// TwinCAT 3 PLC project SchrauberAblauf_SK
// ProgramVersion: 3.1.4024.0
// libraries:
//   Tc2_MC2, * (Beckhoff Automation GmbH)
//   Tc2_Standard, * (Beckhoff Automation GmbH)
//   Tc2_System, * (Beckhoff Automation GmbH)
//   Tc2_Utilities, * (Beckhoff Automation GmbH)
//   Tc3_Module, * (Beckhoff Automation GmbH)
//   UniLib Gruppe 11, * (Beckhoff Automation GmbH & Co. KG)
//   UniNc Gruppe 11, * (Beckhoff Automation GmbH & Co. KG)
//   VisuSymbols,3.5.10.0,System
// project tree:
//   DUTs/ ST_MeldServoSchrauber_1.TcDUT (not stored), ST_ParamSKSServoschrauber.TcDUT (not stored), ST_SKSSchrauberInOut_Vis.TcDUT
//   / GlobalTextList.TcGTLO, PlcTask.TcTTO (not stored), TL_AuswahlSchrauberAblauf.TcTLO, Visualisierungsmanager.TcVMO (not stored)
//   GVLs/ GlobalVar_InOut.TcGVL, GlobalVar_Constant.TcGVL, GlobalVar_NcAchsen.TcGVL, GVL_VISU_SCHRAUBER.TcGVL
//   POUs/10_Funktionen/Diverse/ FB_AchsStartAusf.TcPOU, FB_ErrorCnt.TcPOU (not stored), FB_LogFile_Schrauber.TcPOU, FB_Mittelwert.TcPOU (not stored), FB_OBJ_TimeStamp.TcPOU, FB_Zeitstempel.TcPOU, F_Inbetween.TcPOU (not stored), F_PosZustand.TcPOU
//   POUs/10_Funktionen/History/ FB_StepHistory.TcPOU (not stored)
//   POUs/10_Funktionen/SchraubBearb/Obj/ FB_Obj_Error_Schrauber.TcPOU (not stored), FB_Obj_IOSchlauch.TcPOU
//   POUs/ MAIN.TcPOU, prgMAIN.TcPOU, PRG_Schrauber.TcPOU
//   POUs/SchrauberAblauf/ FB_Schrauber_PnP.TcPOU, FB_Schrauber_PnP_Neu_1.TcPOU
//   POUs/Simulationsprogramm/ FB_Schrauber_Simulation.TcPOU, PRG_Schrauber_Test.TcPOU
//   VISUs/ Frame_Schlauch_Bedien.TcVIS, Frame_Schrauber.TcVIS, Frame_Schrauber_Bedien.TcVIS, Frame_Schrauber_Status.TcVIS, Schrauber_Aufruf.TcVIS

// ---- DUTs/ST_SKSSchrauberInOut_Vis.TcDUT
TYPE ST_SKSSchrauberInOut_Vis :
STRUCT
	I_bTaktFrg						: BOOL;
	I_bTaktStop						: BOOL;
	I_bAuto							: BOOL;
	I_bHand							: BOOL;
	I_bQuittFehler					: BOOL;

	I_bTaktStart					: BOOL;	(*Start Schienenschrauben*)

	I_bGrdstlgSchrEinh				: BOOL;
	I_bZustellZylAusgef				: BOOL;

	I_fSchraubTiefeAuswurf			: LREAL;

	I_fTiefentoleranzPositiv		: LREAL:=1;	(* Z.B. 3 bedeutet, dass von Solltiefe bis + 3mm wir im Ziel liegen *)
	I_fTiefentoleranzNegativ		: LREAL:=0.5;	(* Z.B. 3 bedeutet, dass von Solltiefe bis - 3mm wir im Ziel liegen *)
		
	I_bSchraubeNachschiessen		: BOOL;

	I_bFreigabeAuswerfen			: BOOL;
	
	I_bSchlauchBelegt				:BOOL;
	I_bSchrauberBelegt				:BOOL;
	I_bAuswurfStart					:BOOL;
	I_bVereinzelungStart			:BOOL;
	
	Q_bBusy							: BOOL;
	Q_bDone							: BOOL;
	Q_bError						: BOOL;
	
	Q_nErrorId						: INT;
	Q_bDrehmomentFehler				: BOOL;
	
	Q_bDrehmomentOk					:BOOL;
	
	Q_nActTorque					:LREAL; 	(* Drehmoment ausgabe Mittelwert *)
	Q_nActDepth						:LREAL; 	(* Tiefen ausgabe  *)
	Q_nActVelo						:LREAL;		
	Q_nActPos						:LREAL;
	
	Q_nLastTorque					:LREAL;
	Q_nLastDepth					:LREAL;
	
	Q_nStep							: INT;
	
	Q_strStep						: STRING;
	Q_sStatus						: STRING(255);	//Informationen zu dem aktuellen Ablaufschritt
	
END_STRUCT
END_TYPE

// ---- GVLs/GlobalVar_InOut.TcGVL
{attribute 'Tc2GvlVarNames'}
VAR_GLOBAL
	(* Inputs *)
	bGVLEndlageZyl_1_Eingef	AT %I*: BOOL;
	bGVLEndlageZyl_1_Ausgef	AT %I*: BOOL;
	
	bGVLEndlageZyl_2_Eingef	AT %I*: BOOL;
	bGVLEndlageZyl_2_Ausgef	AT %I*: BOOL;
	
	(* Outputs *)
	bGVLVentil_1_Ausfahr	AT %Q*: BOOL;
	bGVLVentil_1_Einfahr	AT %Q*: BOOL;
	
	bGVLVentil_2_Ausfahr	AT %Q*: BOOL;
	bGVLVentil_2_Einfahr	AT %Q*: BOOL;
	
END_VAR

// ---- GVLs/GlobalVar_Constant.TcGVL
{attribute 'Tc2GvlVarNames'}
VAR_GLOBAL CONSTANT
	cGrundPos								:INT :=1;
	cBearbPos								:INT :=3;
	
	cAxis1261_Schrauber1					:INT := 1;
	cEnc03_Schrauber1						:INT := 2;
	
END_VAR

// ---- GVLs/GlobalVar_NcAchsen.TcGVL
{attribute 'Tc2GvlVarNames'}
VAR_GLOBAL
	
	arrAxis									: ARRAY[1..2] OF AXIS_REF;
	arrNcAchsen								: ARRAY[1..2] OF  TC3_UniLib.ST_NcAchsen;		(* Achtung 1 = Achse / 2= Encoder für Tiefenmessung *)
	arrStartAusf							: ARRAY[1..2] OF FB_AchsStartAusf;
	arrAnstgSchrauberAchse					: ARRAY[1..2] OF FB_AchsKontrlAnstg;
	
	arrBetrartAutomAktiv					:ARRAY[1..2] OF BOOL;
	arrAntrGruppeFrg						:ARRAY[1..2] OF BOOL;
	stParamSKSServoschrauber				:ST_ParamSKSServoschrauber;
	
	objSchlauch								: FB_Obj_IOSchlauch;
	stAchsMeldung							: ST_MeldServoSchrauber_1;					
	bTakt2Langsam							:BOOL;
	
	
	
END_VAR

// ---- GVLs/GVL_VISU_SCHRAUBER.TcGVL
{attribute 'Tc2GvlVarNames'}
VAR_GLOBAL
	stSKSSchrauberInOut_Vis_Schr_1		:ST_SKSSchrauberInOut_Vis;
END_VAR

// ---- POUs/10_Funktionen/Diverse/FB_AchsStartAusf.TcPOU
FUNCTION_BLOCK FB_AchsStartAusf
VAR_INPUT

	I_nAchsNr			:INT;

	I_nSchutzBer		:INT;

	I_bAchseZurGrdP	:BOOL;
	I_bAchseZurArbP	:BOOL;
	I_bAchseStopPos	:BOOL; (*Achse wird gestoppt. Ist nur bei einem aktiven Achsstart ausführbar*)

	I_bAchseFrgGrdP	:BOOL;
	I_bAchseFrgArbP	:BOOL;
	I_bAchseFrgRglP	:BOOL;

	I_bEilSchlAchse	:BOOL;

	I_nStreckeRglP		:INT:= 10;
	I_tDauerAntrFrg	:TIME:= t#1500ms;

	(*ToDo: AchsEinzlStart
			  AchsNachStart
			  AchsNachRegeln
			  AchsOverride	
			  AchsStopp*)

END_VAR
VAR_OUTPUT

	Q_bAchsePosFehl	:BOOL;

	Q_bAchseAktiv		:BOOL;
	Q_bAchseInPos		:BOOL;
	Q_bAchseGestPos	:BOOL;

END_VAR
VAR

	nAchsezurRglP	:BOOL;
	nAchseInRglP	:BOOL;

	nAchseStart		:BOOL;
	nAchseStop		:BOOL;

	tonAntrFrg		:TON;
	
	nStepAchsStop	:INT;

END_VAR

	(*Achs-Fahrauftrag ausführen*)

	IF NOT nAchseInRglP
		AND arrNcAchsen[I_nAchsNr].fPosIstwert < (arrNcAchsen[I_nAchsNr].stAuftrg.fPTP_ZielPos + I_nStreckeRglP)
		AND arrNcAchsen[I_nAchsNr].fPosIstwert > (arrNcAchsen[I_nAchsNr].stAuftrg.fPTP_ZielPos - I_nStreckeRglP)
		AND arrBetrartAutomAktiv[I_nSchutzBer]
			THEN
				nAchsezurRglP:= TRUE;
	END_IF

	IF NOT I_bAchseFrgRglP
		OR I_bAchseZurGrdP
		OR I_bAchseZurArbP
		OR (nAchsezurRglP
		AND Q_bAchseInPos)
		OR I_bEilSchlAchse
		THEN
			nAchsezurRglP:= FALSE;
			nAchseInRglP:= TRUE;
	END_IF

	IF NOT arrNcAchsen[I_nAchsNr].stFreigb.bReglerFrg
		THEN
			nAchseInRglP:= FALSE;
	END_IF

	IF I_bAchseFrgRglP
		AND (arrNcAchsen[I_nAchsNr].fPosIstwert >= (arrNcAchsen[I_nAchsNr].stAuftrg.fPTP_ZielPos + I_nStreckeRglP)
		OR arrNcAchsen[I_nAchsNr].fPosIstwert <= (arrNcAchsen[I_nAchsNr].stAuftrg.fPTP_ZielPos - I_nStreckeRglP))
		(*AND BetrartAutom_aktiv[SchutzBer]*)
			THEN
				Q_bAchsePosFehl:= TRUE;
			ELSE
				Q_bAchsePosFehl:= FALSE;
	END_IF

(**********************************************************************)
(*Achs-Fahrauftrag ausführen*)

	IF I_bAchseZurGrdP
		OR I_bAchseZurArbP
		OR nAchsezurRglP
		THEN
			(*Schleichachse*)
			IF NOT nAchseStart
				AND I_bAchseZurGrdP
				AND (arrNcAchsen[I_nAchsNr].stParam.fGrdstlgPos <= (arrNcAchsen[I_nAchsNr].fPosIstwert + 5)
				AND arrNcAchsen[I_nAchsNr].stParam.fGrdstlgPos >= (arrNcAchsen[I_nAchsNr].fPosIstwert - 5))
				AND I_bEilSchlAchse	(*Fkt. Eil.-Schleichachse (Bremswegfenster)*)
				THEN
					Q_bAchseInPos:= TRUE;
			END_IF
			IF NOT nAchseStart
				AND I_bAchseZurArbP
				AND (arrNcAchsen[I_nAchsNr].stAuftrg.fPTP_ZielPos <= (arrNcAchsen[I_nAchsNr].fPosIstwert + 5)
				AND arrNcAchsen[I_nAchsNr].stAuftrg.fPTP_ZielPos >= (arrNcAchsen[I_nAchsNr].fPosIstwert - 5))
				AND I_bEilSchlAchse	(*Fkt. Eil.-Schleichachse (Bremswegfenster)*)
				THEN
					Q_bAchseInPos:= TRUE;
			END_IF

			IF NOT Q_bAchseInPos
				AND NOT Q_bAchseGestPos
				AND (I_bAchseFrgGrdP OR NOT I_bAchseZurGrdP)
				AND (I_bAchseFrgArbP OR NOT I_bAchseZurArbP)
				AND arrNcAchsen[I_nAchsNr].stAuftrg.bPTP_PosiFrg
				THEN
					nAchseStart:= TRUE;
			END_IF

			IF nAchseStart
				AND I_bAchseStopPos
				THEN
					nAchseStop:= TRUE;
			END_IF
			IF nAchseStart
				THEN
					IF arrNcAchsen[I_nAchsNr].stAuftrg.bPTP_aktiv
					THEN
						Q_bAchseAktiv:= TRUE;
					END_IF
					IF arrNcAchsen[I_nAchsNr].stAuftrg.bPTP_inZiel
					THEN
						Q_bAchseAktiv	:= FALSE;
						Q_bAchseInPos	:= TRUE;
						nAchseStart	 	:= FALSE;
						nAchseStop 	 	:= FALSE;
						
						nStepAchsStop	:= 0;	//JP
					END_IF
					IF arrNcAchsen[I_nAchsNr].stAuftrg.bPTP_gest
					THEN
						Q_bAchseAktiv	:= FALSE;
						Q_bAchseGestPos:= TRUE;
						nAchseStart	 	:= FALSE;
						nAchseStop 	 	:= FALSE;
					END_IF
			END_IF
		ELSE
			Q_bAchseAktiv	:= FALSE;
			Q_bAchseInPos	:= FALSE;
			Q_bAchseGestPos:= FALSE;
			nAchseStart	 	:= FALSE;
			nAchseStop  	:= FALSE;
	END_IF

	(*Achse starten*)	
	IF nAchseStart
		THEN
			IF I_bAchseZurGrdP
			THEN
				arrNcAchsen[I_nAchsNr].stAuftrg.arrPTP_start[cGrundPos]:= tonAntrFrg.Q;
				arrNcAchsen[I_nAchsNr].stAuftrg.arrPTP_start[cBearbPos]:= FALSE;
			ELSIF I_bAchseZurArbP
				OR nAchsezurRglP
			THEN
				arrNcAchsen[I_nAchsNr].stAuftrg.arrPTP_start[cGrundPos]:= FALSE;
				arrNcAchsen[I_nAchsNr].stAuftrg.arrPTP_start[cBearbPos]:= tonAntrFrg.Q;
				
				nStepAchsStop	:= 1;	//JP
			END_IF
			arrNcAchsen[I_nAchsNr].stAuftrg.bPTP_stop:= nAchseStop;
		ELSE
			arrNcAchsen[I_nAchsNr].stAuftrg.arrPTP_start[cGrundPos]:= FALSE;
			arrNcAchsen[I_nAchsNr].stAuftrg.arrPTP_start[cBearbPos]:= FALSE;
			arrNcAchsen[I_nAchsNr].stAuftrg.bPTP_stop:= FALSE;
			
		//JP
		CASE nStepAchsStop OF
			 0: //keine Achsbewegung vorhanden
				 arrNcAchsen[I_nAchsNr].stAuftrg.bPTP_AutoStop:= FALSE;
			
			 1: // Achsen Stoppen, wenn keine Automatik aktiv 
				IF NOT arrBetrartAutomAktiv[I_nSchutzBer]
				THEN
					arrNcAchsen[I_nAchsNr].stAuftrg.bPTP_AutoStop	:= TRUE;
					nStepAchsStop	:= 2;
				ELSE
					arrNcAchsen[I_nAchsNr].stAuftrg.bPTP_AutoStop	:= FALSE;					
				END_IF
			 
			 2: // Achsen ist gestoppt 
				IF arrNcAchsen[I_nAchsNr].stAuftrg.bPTP_gest
					OR arrBetrartAutomAktiv[I_nSchutzBer]	 
					OR I_bAchseZurGrdP // wird z.B. bei Achsfehlern benötigt
				THEN
					arrNcAchsen[I_nAchsNr].stAuftrg.bPTP_AutoStop	:= FALSE;
    				nStepAchsStop	:= 0;
				END_IF
		END_CASE
	END_IF

	tonAntrFrg (
		IN:= arrAntrGruppeFrg[I_nSchutzBer],
		PT:= I_tDauerAntrFrg
		);

END_FUNCTION_BLOCK

// ---- POUs/10_Funktionen/SchraubBearb/Obj/FB_Obj_IOSchlauch.TcPOU
FUNCTION_BLOCK FB_Obj_IOSchlauch
VAR_INPUT
	 
	I_bFrgNachladen				: BOOL;	(* Schrauber -> *)
	I_bVereinzelungskontrolle	: BOOL;	(* Schrauber -> *)
	I_bSotiertopfEin				: BOOL;	(* Schrauber -> *)

	I_bSchrauberBelegt			: BOOL;	(* Rütteltopf -> *)
	I_bSchlauchBelegt				: BOOL;	(* Rütteltopf -> *)
	I_bSchrAuswurfStart			: BOOL;	(* Rütteltopf -> *)

	I_bTasteVereinzelung			: BOOL;	(*am Rütteltopf*)
	I_bTasteNachruetteln			: BOOL;

	I_bNachladenaktiv 			: BOOL := FALSE;

END_VAR
VAR_OUTPUT
END_VAR
VAR
END_VAR

;

END_FUNCTION_BLOCK

// ---- POUs/10_Funktionen/Diverse/FB_LogFile_Schrauber.TcPOU
FUNCTION_BLOCK FB_LogFile_Schrauber
VAR_INPUT
	I_bStart			: BOOL;	

	I_sDateipfad	: T_MaxString;
	I_sDateiname	: T_MaxString;
	I_sUeberschrift: T_MaxString;
(*	I_sZeile			: T_MaxString;*)

	I_sFehler1		: STRING;
	I_sFehler2		: STRING;
	I_sFehler3		: STRING;
	I_sFehler4		: STRING;
	I_sFehler5		: STRING;
	I_sFehler6		: STRING;
	I_sFehler7		: STRING;
	I_sFehler8		: STRING;
	I_sFehler9		: STRING;

	I_sBarcode		: STRING(19);

	I_bFehler1		: BOOL;
	I_bFehler2		: BOOL;
	I_bFehler3		: BOOL;
	I_bFehler4		: BOOL;
	I_bFehler5		: BOOL;
	I_bFehler6		: BOOL;
	I_bFehler7		: BOOL;
	I_bFehler8		: BOOL;
	I_bFehler9		: BOOL;

	I_nAnzahlVerschraubungen		: INT;

	I_tSchraubzeit						: TIME;
	I_fSchraubtiefe					: LREAL;
	I_fDrehmoment						: LREAL;
		
	I_fbZeitstempel	: FB_Zeitstempel;				(*Zeitstempelbaustein zum Schreiben der Logdatei*)

END_VAR
VAR_OUTPUT
	Q_bDone		: BOOL;
END_VAR
VAR
	nStep			: INT;
	sPfadname	: T_MaxString;
	sZeile		: T_MaxString;
	fbFindFile	: FB_EnumFindFileEntry;
	fbFileOpen 	: FB_FileOpen;
	fbFileWrite : FB_FileWrite;
	fbFileClose	: FB_FileClose;
	
	sLogZeile	: T_MaxString;	

END_VAR

a_LogZeile();

CASE nStep OF

0: (*INIT*)
	fbFileOpen(bExecute := FALSE);
	fbFindFile(bExecute := FALSE);
	fbFileWrite(bExecute := FALSE);
	fbFileClose(bExecute := FALSE);
	sPfadname	:= '';
	Q_bDone		:= FALSE;
	IF I_bStart
		AND sLogZeile <> ''
	THEN
		sPfadname :=CONCAT(CONCAT(CONCAT(I_sDateipfad,'\'),I_sDateiname),'.csv');
		nStep := 5;
	END_IF


5: (*Check ob Datei vorhanden ist*)
	fbFindFile(
		sNetId		:= , 
		sPathName	:= sPfadname, 
		eCmd			:= , 
		bExecute		:= TRUE, 
		tTimeout		:= T#2S, 
		bBusy			=> , 
		bError		=> , 
		nErrID		=> , 
		bEOE			=> , 
		stFindFile	=> );
	
	IF NOT fbFindFile.bBusy
		AND NOT fbFindFile.bError
	THEN
		nStep:= 10;
	END_IF


10: (* Öffne Datei*)
	fbFileOpen(
		sNetId		:= , 
		sPathName	:= sPfadname, 
		nMode			:= FOPEN_MODEAPPEND OR FOPEN_MODEPLUS, 
		ePath			:= PATH_GENERIC , 
		bExecute		:= TRUE, 
		tTimeout		:= T#2S, 
		bBusy			=> , 
		bError		=> , 
		nErrId		=> , 
		hFile			=> );
		
	IF NOT fbFileOpen.bBusy
		AND NOT fbFileOpen.bError
	THEN
		IF fbFindFile.stFindFile.sFileName <> ''
		THEN
			nStep := 20;
		ELSE
			nStep:= 13;
		END_IF
	END_IF
	

13: (* Schreibe Überschrift*)
	fbFileWrite(
		sNetId		:= , 
		hFile			:= fbFileOpen.hFile, 
		pWriteBuff	:= ADR(I_sUeberschrift), 
		cbWriteLen	:= LEN(I_sUeberschrift), 
		bExecute		:= TRUE, 
		tTimeout		:= T#2S, 
		bBusy			=> , 
		bError		=> , 
		nErrId		=> , 
		cbWrite		=> );
		
	IF NOT fbFileWrite.bBusy
		AND NOT fbFileWrite.bError
	THEN
		nStep:= 14;
	END_IF

14:
	fbFileWrite(
		bExecute		:= FALSE); 
	nStep:= 20;
	

20: (* Schreibe Datei*)
	sZeile:= CONCAT(sLogZeile,'$R');
	fbFileWrite(
		sNetId		:= , 
		hFile			:= fbFileOpen.hFile, 
		pWriteBuff	:= ADR(sZeile), 
		cbWriteLen	:= LEN(sZeile), 
		bExecute		:= TRUE, 
		tTimeout		:= T#2S, 
		bBusy			=> , 
		bError		=> , 
		nErrId		=> , 
		cbWrite		=> );
		
	IF NOT fbFileWrite.bBusy
		AND NOT fbFileWrite.bError
	THEN
		nStep:= 30;
	END_IF
	

30: (* Schließe Datei*)
	fbFileClose(
		sNetId	:= , 
		hFile		:= fbFileOpen.hFile, 
		bExecute	:= TRUE, 
		tTimeout	:= T#2S, 
		bBusy		=> , 
		bError	=> , 
		nErrId	=> );
		
	IF NOT fbFileClose.bBusy
		AND NOT fbFileClose.bError
	THEN
		nStep:= 40;
	END_IF
	

40: (* Melde DONE*)
	Q_bDone := TRUE;
	IF NOT I_bStart
	THEN
		nStep:= 0;
	END_IF

END_CASE

ACTION a_LogZeile:
sLogZeile := '';

sLogZeile:= CONCAT(sLogZeile,WORD_TO_STRING(prgMAIN.fbZeitstempel.Q_objTimestamp.nJahr));
sLogZeile:= CONCAT(sLogZeile,'-');
IF prgMAIN.fbZeitstempel.Q_objTimestamp.nMonat < 10
THEN
sLogZeile:= CONCAT(sLogZeile,'0');
END_IF
sLogZeile:= CONCAT(sLogZeile,WORD_TO_STRING(prgMAIN.fbZeitstempel.Q_objTimestamp.nMonat));
sLogZeile:= CONCAT(sLogZeile,'-');
IF prgMAIN.fbZeitstempel.Q_objTimestamp.nTag < 10
THEN
sLogZeile:= CONCAT(sLogZeile,'0');
END_IF
sLogZeile:= CONCAT(sLogZeile,WORD_TO_STRING(prgMAIN.fbZeitstempel.Q_objTimestamp.nTag));
sLogZeile:= CONCAT(sLogZeile,'-');
IF prgMAIN.fbZeitstempel.Q_objTimestamp.nStunde < 10
THEN
sLogZeile:= CONCAT(sLogZeile,'0');
END_IF
sLogZeile:= CONCAT(sLogZeile,WORD_TO_STRING(prgMAIN.fbZeitstempel.Q_objTimestamp.nStunde));
sLogZeile:= CONCAT(sLogZeile,':');
IF prgMAIN.fbZeitstempel.Q_objTimestamp.nMinute < 10
THEN
sLogZeile:= CONCAT(sLogZeile,'0');
END_IF
sLogZeile:= CONCAT(sLogZeile,WORD_TO_STRING(prgMAIN.fbZeitstempel.Q_objTimestamp.nMinute));
sLogZeile:= CONCAT(sLogZeile,':');
IF prgMAIN.fbZeitstempel.Q_objTimestamp.nSekunde < 10
THEN
sLogZeile:= CONCAT(sLogZeile,'0');
END_IF
sLogZeile:= CONCAT(sLogZeile,WORD_TO_STRING(prgMAIN.fbZeitstempel.Q_objTimestamp.nSekunde));
sLogZeile:= CONCAT(sLogZeile,';');

sLogZeile:= CONCAT(sLogZeile,INT_TO_STRING(I_nAnzahlVerschraubungen));
sLogZeile:= CONCAT(sLogZeile,';');

sLogZeile:= CONCAT(sLogZeile,TIME_TO_STRING(I_tSchraubzeit));
sLogZeile:= CONCAT(sLogZeile,';');

sLogZeile:= CONCAT(sLogZeile,TO_STRING(I_fDrehmoment));
sLogZeile:= CONCAT(sLogZeile,';');

sLogZeile:= CONCAT(sLogZeile,TO_STRING(I_fSchraubtiefe));
sLogZeile:= CONCAT(sLogZeile,';');

sLogZeile:= CONCAT(sLogZeile, I_sBarcode);
sLogZeile:= CONCAT(sLogZeile,';');

IF I_bFehler1
THEN
	sLogZeile:= CONCAT(sLogZeile,I_sFehler1);
END_IF
IF I_bFehler2
THEN
	sLogZeile:= CONCAT(sLogZeile,I_sFehler2);
END_IF
IF I_bFehler3
THEN
	sLogZeile:= CONCAT(sLogZeile,I_sFehler3);
END_IF
IF I_bFehler4
THEN
	sLogZeile:= CONCAT(sLogZeile,I_sFehler4);
END_IF
IF I_bFehler5
THEN
	sLogZeile:= CONCAT(sLogZeile,I_sFehler5);
END_IF
IF I_bFehler6
THEN
	sLogZeile:= CONCAT(sLogZeile,I_sFehler6);
END_IF
IF I_bFehler7
THEN
	sLogZeile:= CONCAT(sLogZeile,I_sFehler7);
END_IF
IF I_bFehler8
THEN
	sLogZeile:= CONCAT(sLogZeile,I_sFehler8);
END_IF
IF I_bFehler9
THEN
	sLogZeile:= CONCAT(sLogZeile,I_sFehler9);
END_IF
sLogZeile:= CONCAT(sLogZeile,';');
END_ACTION

END_FUNCTION_BLOCK

// ---- POUs/10_Funktionen/Diverse/FB_Zeitstempel.TcPOU
FUNCTION_BLOCK FB_Zeitstempel
	(******************************************************************)
	(*	Version history																*)
	(*	Date				:	17/01/2002												*)
	(*	Version			:	2.0.0														*)
 	(*	Created under	:	2.7.0	(Build 405)										*)
	(*	Author			:	Torsten Schulz											*)
	(******************************************************************)
	(*	History			:																*)
	(*	Irgendwann mal	-	Erste Version											*)
	(*	17.01.2002		- 	Zeitbasis durch Vielfaches der Zykluszeit.	*)
	(*							Synchronisierung 1xproSekunde, hSec werden	*)
	(*							durch Plc-Task incrementiert.						*)
	(******************************************************************)
VAR_INPUT
	I_bHochkomma 		:	BOOL;					(* Jeweils Datum und Uhrzeit in Hochkommata *)
	I_bSemikolon		:	BOOL;					(* Datum- Uhrzeit-Treuung mit Semikolon, Standard ist Bindestrich *)
END_VAR
VAR_OUTPUT
	Q_objTimestamp	:	FB_OBJ_TimeStamp;			(* Alle Ausgangswerte zusammengefasst *)
END_VAR
VAR
	bInitOk			:	BOOL;						(* Für einmaliges Lesen der Zykluszeit *)
	nSPS_Taskzeit	:	UINT;						(* Ermittelte SPS-Zykluszeit *)
	fbTaskIndex		:	GETCURTASKINDEX;		(* Instanz zur Ermittlung des SPS-Task		*)
	nCounter			:	UDINT;					(* Zähler für hSec-Äquivalent durch Zykluszeit *)
	rtrigStart		:	R_TRIG;					(* Trigger zum Start der Formatierung nach neuer Zeitlesung *)
	nSec				:	WORD;						(* Hilfsvariable für hSec Darstellung *)
	sQ1				:	STRING;					(* Hilfvariable zur Formaterzeugung *)

	sHochkomma		:	STRING(2);				(* Hochkomma-Platzhalter *)
	sSemikolon		:	STRING(3);				(* Semikolon-Platzhalter *)
	stTimeStr		:	TimeStruct;				(* Structur zum Lesen der Zeit *)
	fbgettime		:	NT_GetTime;				(* Instanz zum Lesen der Zeit *)
END_VAR

	(****************************************************************************************)
	(* Lesen der Zykluszeit des Task *)
	IF NOT bInitOk
	THEN
		(* Aktuellen SPS-Task ermitteln *)
		fbTaskIndex();

		(* Ermitteln der SPS-Zykluszeit im ms*)
		nSPS_Taskzeit:=
			UDINT_TO_UINT(_TaskInfo[fbTaskIndex.INDEX].cycleTime / 10000);

		bInitOk	:= TRUE;
	END_IF

	(****************************************************************************************)
	IF I_bHochkomma
	THEN
		sHochkomma := '"';
	ELSE
		sHochkomma := '';
	END_IF

	IF I_bSemikolon
	THEN
		sSemikolon := ';';
	ELSE
		sSemikolon := ' - ';
	END_IF

	nCounter := nCounter + nSPS_Taskzeit;
	IF	nCounter >= (1000)
	THEN
		nCounter := 0;
	END_IF

	fbgettime(Start := (nCounter = 0));

	rtrigStart(
		Clk	:=	NOT fbgettime.BUSY);

	IF	rtrigStart.Q
	THEN

		(****************************************************************************************)
		(* Zeitstring holen *)
		stTimeStr := fbgettime.TimeStr;

		sQ1 := '';

		(****************************************************************************************)
		(* ggf Hochkomma wenn CSV-Datei *)
		sQ1 := CONCAT(sQ1,sHochkomma);

		(****************************************************************************************)
		(* Tag *)
		IF stTimeStr.wDay < 10
		THEN
			sQ1 := CONCAT(sQ1,'0');
		END_IF
		sQ1 := CONCAT(sQ1,WORD_TO_STRING(stTimeStr.wDay));
		sQ1 := CONCAT(sQ1,'.');

		Q_objTimestamp.nTag				:=	stTimeStr.wDay;
		Q_objTimestamp.nTagDerWoche	:=	stTimeStr.wDayOfWeek;

		(****************************************************************************************)
		(* Monat *)
		IF stTimeStr.wMonth < 10
		THEN
			sQ1 := CONCAT(sQ1,'0');
		END_IF
		sQ1 := CONCAT(sQ1,WORD_TO_STRING(stTimeStr.wMonth));
		sQ1 := CONCAT(sQ1,'.');

		Q_objTimestamp.nMonat	:=	stTimeStr.wMonth;

		(****************************************************************************************)
		(* Jahr *)
		sQ1 := CONCAT(sQ1,WORD_TO_STRING(stTimeStr.wYear));

		Q_objTimestamp.nJahr	:=	stTimeStr.wYear;

		(****************************************************************************************)
		(* ggf Hochkomma wenn CSV-Datei *)
		sQ1 := CONCAT(sQ1,sHochkomma);

		(****************************************************************************************)
		(* Trennung *)
		sQ1 := CONCAT(sQ1,sSemikolon);

		(****************************************************************************************)
		(* ggf Hochkomma wenn CSV-Datei *)
		sQ1 := CONCAT(sQ1,sHochkomma);

		(****************************************************************************************)
		(* Stunde *)
		IF stTimeStr.wHour < 10
		THEN
			sQ1 := CONCAT(sQ1,'0');
		END_IF

		sQ1 := CONCAT(sQ1,WORD_TO_STRING(stTimeStr.wHour));
		sQ1 := CONCAT(sQ1,':');

		Q_objTimestamp.nStunde	:=	stTimeStr.wHour;

		(****************************************************************************************)
		(* Minute *)
		IF stTimeStr.wMinute < 10
		THEN
			sQ1 := CONCAT(sQ1,'0');
		END_IF

		sQ1 := CONCAT(sQ1,WORD_TO_STRING(stTimeStr.wMinute));
		sQ1 := CONCAT(sQ1,':');

		Q_objTimestamp.nMinute	:=	stTimeStr.wMinute;

		(****************************************************************************************)
		(* Sekunde *)
		IF stTimeStr.wSecond < 10
		THEN
			sQ1 := CONCAT(sQ1,'0');
		END_IF

		sQ1 := CONCAT(sQ1,WORD_TO_STRING(stTimeStr.wSecond));
		sQ1 := CONCAT(sQ1,':');

		Q_objTimestamp.nSekunde	:=	stTimeStr.wSecond;
		nSec		:= 0;
	ELSE
		nSec	:=	nSec + nSPS_Taskzeit;

		IF	nSec >= 1000
		THEN
			nSec	:= 0;
		END_IF

		IF 	(nSec < 100)
			AND (nSec > 9)
		THEN
			Q_objTimestamp.sQ := CONCAT('0', WORD_TO_STRING(nSec));
		ELSIF nSec < 10
		THEN
			Q_objTimestamp.sQ := CONCAT('00', WORD_TO_STRING(nSec));
		ELSE
			Q_objTimestamp.sQ := WORD_TO_STRING(nSec);
		END_IF

		IF LEN(sQ1) > 0
		THEN
			Q_objTimestamp.sQ := CONCAT(sQ1,Q_objTimestamp.sQ);

			(****************************************************************************************)
			(* ggf Hochkomma wenn CSV-Datei *)
			Q_objTimestamp.sQ := CONCAT(Q_objTimestamp.sQ,sHochkomma);

		END_IF
	END_IF

END_FUNCTION_BLOCK

// ---- POUs/10_Funktionen/Diverse/FB_OBJ_TimeStamp.TcPOU
{attribute 'pack_mode' := '1'}
FUNCTION_BLOCK FB_OBJ_TimeStamp
VAR_INPUT
	sQ					:	STRING;				(* Zeitstempel *)
	nStunde			:	WORD;					(* Stunde als Dezimalwert *)
	nMinute			:	WORD;					(* Minute als Dezimalwert *)
	nSekunde			:	WORD;					(* Sekunde als Dezimalwert *)
	nTag				:	WORD;					(* Tag als Dezimalwert *)
	nMonat			:	WORD;					(* Monat als Dezimalwert *)
	nJahr				:	WORD;					(* Jahr als Dezimalwert *)
	nTagDerWoche	:	WORD;					(* Tag der Woche  als Dezimalwert *)
END_VAR
VAR_OUTPUT
END_VAR
VAR
END_VAR

;

END_FUNCTION_BLOCK

// ---- POUs/prgMAIN.TcPOU
PROGRAM prgMAIN
VAR
	(* Sonstiges *)
	fbZeitstempel	:	FB_Zeitstempel;
END_VAR


	fbZeitstempel();

END_PROGRAM

// ---- POUs/10_Funktionen/Diverse/F_PosZustand.TcPOU
FUNCTION F_PosZustand : STRING(80)
VAR_INPUT
	I_sString	:STRING;
	I_nStep 		:INT;
	I_sStep 		:STRING;
END_VAR
VAR
	stemp 	:STRING;
END_VAR

	stemp := 'nStep : ' (*CONCAT(I_string,' - nStep : ');*);
	stemp := CONCAT(stemp,INT_TO_STRING(I_nStep));
	stemp := CONCAT(stemp,' - ');
	stemp := CONCAT(stemp,I_sStep);


	F_PosZustand := stemp;

END_FUNCTION

// ---- POUs/MAIN.TcPOU
PROGRAM MAIN
VAR

END_VAR

PRG_Schrauber();

END_PROGRAM

// ---- POUs/PRG_Schrauber.TcPOU
PROGRAM PRG_Schrauber
VAR
	fbSchrauber_PnP_Original	:FB_Schrauber_PnP;
	fbSchrauber_PnP_Entwickel	:FB_Schrauber_PnP_Neu_1;
	
	nAchsId : INT;
	
	iAuswSchrauberMode	:INT := 0;	(* 0 = Original Ablauf | 1 = Versuch Ablauf *)
	
END_VAR

ac01_AchsAnstrg();

CASE iAuswSchrauberMode OF
0:	ac00_Init();	(* Reset beide Abläufe *)
1:	ac10_OriginalSchrauberAblauf();
2:	ac11_EntwickelungSchrauberAblauf();
END_CASE

ACTION ac00_Init:
(* RESET *)


fbSchrauber_PnP_Original(
	I_bResetTeststation := 			TRUE,
	IQ_fbObjSchlauch:= 				objSchlauch, 
	IQ_stMeldung:= 					stAchsMeldung);
	
fbSchrauber_PnP_Entwickel(
	I_bResetTeststation := 			TRUE,
	IQ_fbObjSchlauch:= 				objSchlauch, 
	IQ_stMeldung:= 					stAchsMeldung);
END_ACTION

ACTION ac01_AchsAnstrg:

(*=============================================================================================*)
(* Achsanschaltung Global für alle Schrauberabläufe Gleich*)
(*=============================================================================================*)
arrBetrartAutomAktiv[1] := TRUE;
arrAntrGruppeFrg[1] := TRUE;
arrAntrGruppeFrg[2] := TRUE;

nAchsId	:= cAxis1261_Schrauber1;
	
(*=============================================================================================*)
(* NC Achse*)
arrNcAchsen[cAxis1261_Schrauber1].stFreigb.bAntrbEinFrg				:= TRUE;
arrNcAchsen[cAxis1261_Schrauber1].stStatus.bAchseBTB				:= TRUE;	(* Muss noch gemacht werden *)
arrNcAchsen[cAxis1261_Schrauber1].stFreigb.bVorschFrg				:= TRUE;
arrNcAchsen[cAxis1261_Schrauber1].stFreigb.bSensEndlNeg				:= TRUE;
arrNcAchsen[cAxis1261_Schrauber1].stFreigb.bSensEndlPos				:= TRUE;
arrNcAchsen[cAxis1261_Schrauber1].stEinAusG.I_nDigitaleEingaenge.3 	:= TRUE;
arrNcAchsen[cAxis1261_Schrauber1].stEinAusG.I_nDigitaleEingaenge.4	:= TRUE;
arrNcAchsen[cAxis1261_Schrauber1].stAuftrg.bPTP_verz				:= FALSE;
arrNcAchsen[cAxis1261_Schrauber1].stFreigb.fOverride				:= 10;
arrNcAchsen[cAxis1261_Schrauber1].stParam.fEilgGeschw				:= 6000;

(*=============================================================================================*)	
(* Schraubmotor *)
arrAnstgSchrauberAchse[1](
		IQ_stAchse 			:= arrNcAchsen[cAxis1261_Schrauber1],
		IQ_fbAxisRef 		:= arrAxis[cAxis1261_Schrauber1],
		);
(*=============================================================================================*)			
(* Encoder*)									
arrAnstgSchrauberAchse[2](
		IQ_stAchse 			:= arrNcAchsen[cEnc03_Schrauber1],
		IQ_fbAxisRef 		:= arrAxis[cEnc03_Schrauber1],
		);
(*=============================================================================================*)			
(* Ohne Softwareendlagen *)
arrNcAchsen[cAxis1261_Schrauber1].stParam.bOhnSoftEndl:= TRUE;
END_ACTION

ACTION ac10_OriginalSchrauberAblauf:
(*=============================================================================================*)	
(* Originaler SKS-Schrauberablauf von FA Beckhoff Automation- gesichert aus Band222
	Datum: 	11.09.2025
	Author:	N.Kersting/ T.Hinz	 *)
(*=============================================================================================*)	

(*=============================================================================================*)
(* Parameter *)
stParamSKSServoschrauber.fStartDrehzahl				:= 10;
stParamSKSServoschrauber.fParam_Solldrehzahl		:= 40;
stParamSKSServoschrauber.fParam_Sollmoment			:= 1.4;
stParamSKSServoschrauber.fParam_Sollschraubtiefe	:= -4;
stParamSKSServoschrauber.fParam_Umschalttiefe		:= 2;
stParamSKSServoschrauber.tParam_ZeitdAuswurfSchr	:= T#2S;
stParamSKSServoschrauber.tParam_ZeitdSchraubhubSchr	:= T#2S;
stParamSKSServoschrauber.tParam_ZeitdSchraubTakt	:= T#10S;
stParamSKSServoschrauber.tParam_ZeitdZustellhubSchr	:= T#2S;

(*=============================================================================================*)	
(* Achsstart *)
arrStartAusf[cAxis1261_Schrauber1](
	I_nAchsNr			:= cAxis1261_Schrauber1,
	I_nSchutzBer		:= 1,
	I_bAchseFrgGrdP		:=	TRUE,
	I_bAchseFrgArbP		:= TRUE,
	I_bAchseFrgRglP		:= FALSE,
	I_bAchseStopPos		:= 	fbSchrauber_PnP_Original.Q_bSchrHalt,
	I_nStreckeRglP		:= 2);
	
arrNcAchsen[cAxis1261_Schrauber1].stAuftrg.bPTP_halt	:= fbSchrauber_PnP_Original.Q_bSchrHalt;

(*=============================================================================================*)
(* Achsansteurung *)
IF fbSchrauber_PnP_Original.Q_bModuloBetrArt
THEN
	arrAnstgSchrauberAchse[1].I_nBetrArt	:= 1;
ELSE
	arrAnstgSchrauberAchse[1].I_nBetrArt	:= 0;
END_IF

(*=============================================================================================*)	
(* Drehmoment *)
arrNcAchsen[cAxis1261_Schrauber1].stEinAusG.Q_nDrehmomentGrenzwert := fbSchrauber_PnP_Original.Q_nTorque;

(*=============================================================================================*)	
(* Reset *)
arrNcAchsReset[cAxis1261_Schrauber1]:= fbSchrauber_PnP_Original.Q_bAxisReset;

(*=============================================================================================*)	
(* Alter Baustein *)
fbSchrauber_PnP_Original(
	I_bResetTeststation := 			FALSE,
	I_bTaktFrg:= 					stSKSSchrauberInOut_Vis_Schr_1.I_bTaktFrg, 
	I_bTaktStop:= 					stSKSSchrauberInOut_Vis_Schr_1.I_bTaktStop, 
	I_bQuittFehler:= 				stSKSSchrauberInOut_Vis_Schr_1.I_bQuittFehler, 
	I_bSchutzbereichOK:= 			TRUE, 
	I_bTaktStart:= 					stSKSSchrauberInOut_Vis_Schr_1.I_bTaktStart, 
	I_bGrdstlgSchrEinh:= 			bGVLEndlageZyl_1_Eingef (*OR stSKSSchrauberInOut_Vis_Schr_1.I_bGrdstlgSchrEinh*), 	(* Achtung muss nachher wieder weggenommen werden, wenn der Physische aufbau da ist !!!!!*)
	I_bZustellZylAusgef:= 			bGVLEndlageZyl_2_Ausgef (*OR stSKSSchrauberInOut_Vis_Schr_1.I_bZustellZylAusgef*), 	(* Achtung muss nachher wieder weggenommen werden, wenn der Physische aufbau da ist !!!!!*)
	I_fSchraubTiefeAuswurf:= 		, 
	I_fTiefentoleranzPositiv:= 		, 
	I_fTiefentoleranzNegativ:= 		, 
	I_nAchsId:= 					cAxis1261_Schrauber1, 
	I_nEncId:= 						cEnc03_Schrauber1, 
	I_stParam:= 					stParamSKSServoschrauber, 
	I_tAutoQuit:= 					, 
	I_bSchraubeNachschiessen:=		 , 
	I_bReferenzfahrtAktiv:= 		, 
	I_bFreigabeAuswerfen:= 			, 
	I_sDateipfad:= 					, 
	I_bSchrauberLogOn:= 			, 
	I_nMotorHersteller:=			 1, 
	I_bHuettenSchr:= 				, 
	Q_bBusy=> 						stSKSSchrauberInOut_Vis_Schr_1.Q_bBusy, 
	Q_bDone=>						stSKSSchrauberInOut_Vis_Schr_1.Q_bDone ,	 
	Q_bError=>						stSKSSchrauberInOut_Vis_Schr_1.Q_bError , 
	Q_sPosZustand=> , 
	Q_bGrundstellungAktiv=> , 
	Q_bGrundstellungOk=> , 
	Q_bSchraubHub=> , 
	Q_bSchrAuswurf=> , 
	Q_bSchrHalt=> , 
	Q_nTorque=> , 
	Q_bAxisReset=> , 
	Q_nErrorId=> 					stSKSSchrauberInOut_Vis_Schr_1.Q_nErrorId, 
	Q_bDrehmomentFehler=> 			stSKSSchrauberInOut_Vis_Schr_1.Q_bDrehmomentFehler, 
	Q_bTuerFreigabe=> , 
	Q_nStep=> 						stSKSSchrauberInOut_Vis_Schr_1.Q_nStep, 
	Q_strStep=> , 
	Q_bModuloBetrArt=> , 
	Q_sStatus=> 					stSKSSchrauberInOut_Vis_Schr_1.Q_sStatus, 
	IQ_fbObjSchlauch:= 				objSchlauch, 
	IQ_stMeldung:= 					stAchsMeldung);	
	
(*=============================================================================================*)	
(* Schlauch belegung *)
objSchlauch.I_bSchlauchBelegt		:=	stSKSSchrauberInOut_Vis_Schr_1.I_bSchlauchBelegt;
objSchlauch.I_bSchrauberBelegt		:=	stSKSSchrauberInOut_Vis_Schr_1.I_bSchrauberBelegt;
objSchlauch.I_bTasteVereinzelung	:=	stSKSSchrauberInOut_Vis_Schr_1.I_bVereinzelungStart;
objSchlauch.I_bSchrAuswurfStart		:=	stSKSSchrauberInOut_Vis_Schr_1.I_bAuswurfStart;

(*=============================================================================================*)	
(* Visu Übergabe *)
stSKSSchrauberInOut_Vis_Schr_1.Q_nActVelo	:=	arrNcAchsen[cAxis1261_Schrauber1].fVeloIstwert;
stSKSSchrauberInOut_Vis_Schr_1.Q_nActPos	:=	arrNcAchsen[cAxis1261_Schrauber1].fPosIstwert;
stSKSSchrauberInOut_Vis_Schr_1.Q_nActDepth	:=	arrNcAchsen[cEnc03_Schrauber1].fPosIstwert;


(*=============================================================================================*)	
(* Output Übergabe *)

bGVLVentil_1_Ausfahr:=		fbSchrauber_PnP_Original.Q_bSchraubHub;
bGVLVentil_1_Einfahr:=		NOT fbSchrauber_PnP_Original.Q_bSchraubHub;

bGVLVentil_2_Ausfahr:=		fbSchrauber_PnP_Original.Q_bSchrAuswurf;
bGVLVentil_2_Einfahr:=		NOT fbSchrauber_PnP_Original.Q_bSchrAuswurf;
END_ACTION

ACTION ac11_EntwickelungSchrauberAblauf:
(*=============================================================================================*)	
(* Neu Entwickelter Versuchs Ablauf nach Nobilia Vorgabe 
	aus Dokument vom 22.03.2023 Besprechungsprotokoll Ablaufbeschreibung SKS Schrauber.
	
	Datum: 	11.09.2025
	Author:	N.Kersting/ T.Hinz	 *)
(*=============================================================================================*)	

(*=============================================================================================*)	
(* Parameter *)
stParamSKSServoschrauber.fStartDrehzahl				:= 10;
stParamSKSServoschrauber.fParam_Solldrehzahl		:= 40;
stParamSKSServoschrauber.fParam_Sollmoment			:= 1.4;
stParamSKSServoschrauber.fParam_Sollschraubtiefe	:= -4;
stParamSKSServoschrauber.fParam_Umschalttiefe		:= 2;
stParamSKSServoschrauber.tParam_ZeitdAuswurfSchr	:= T#2S;
stParamSKSServoschrauber.tParam_ZeitdSchraubhubSchr	:= T#2S;
stParamSKSServoschrauber.tParam_ZeitdSchraubTakt	:= T#10S;
stParamSKSServoschrauber.tParam_ZeitdZustellhubSchr	:= T#2S;

(*=============================================================================================*)	
(* Achsstart *)
arrStartAusf[cAxis1261_Schrauber1](
	I_nAchsNr			:= cAxis1261_Schrauber1,
	I_nSchutzBer		:= 1,
	I_bAchseFrgGrdP		:=	TRUE,
	I_bAchseFrgArbP		:= TRUE,
	I_bAchseFrgRglP		:= FALSE,
	I_bAchseStopPos		:= 	fbSchrauber_PnP_Entwickel.Q_bSchrHalt,
	I_nStreckeRglP		:= 2);

arrNcAchsen[cAxis1261_Schrauber1].stAuftrg.bPTP_halt	:= fbSchrauber_PnP_Entwickel.Q_bSchrHalt;

(*=============================================================================================*)
(* Achsansteurung *)
arrAnstgSchrauberAchse[1].I_nBetrArt	:= 1;	

(*=============================================================================================*)	
(* Drehmoment *)
arrNcAchsen[cAxis1261_Schrauber1].stEinAusG.Q_nDrehmomentGrenzwert := fbSchrauber_PnP_Entwickel.Q_nTorque;
	
(*=============================================================================================*)	
(* Reset *)
arrNcAchsReset[cAxis1261_Schrauber1]:= fbSchrauber_PnP_Entwickel.Q_bAxisReset;

(*=============================================================================================*)	
(* Neuer Ablauf *)
fbSchrauber_PnP_Entwickel(
	I_bResetTeststation := 			FALSE,
	I_bTaktFrg:= 					stSKSSchrauberInOut_Vis_Schr_1.I_bTaktFrg, 
	I_bTaktStop:= 					stSKSSchrauberInOut_Vis_Schr_1.I_bTaktStop, 
	I_bAuto:= , 
	I_bHand:= , 
	I_bQuittFehler:= 				stSKSSchrauberInOut_Vis_Schr_1.I_bQuittFehler, 
	I_bGrundstellung:= , 
	I_bSchutzbereichOK:= 			TRUE, 
	I_bTaktStart:= 					stSKSSchrauberInOut_Vis_Schr_1.I_bTaktStart, 
	I_bTaktStartHalb:= , 
	I_bGrdstlgSchrEinh:= , 
	I_bZustellZylAusgef:= , 
	I_fSchraubTiefeAuswurf:= , 
	I_fTiefentoleranzPos:= , 
	I_fTiefentoleranzNeg:= , 
	I_nAchsId:= 					cAxis1261_Schrauber1, 
	I_nEncId:= 						cEnc03_Schrauber1, 
	I_stParam:= 					stParamSKSServoschrauber, 
	I_tAutoQuit:= , 
	I_bSchraubeNachschiessen:= , 
	I_bReferenzfahrtAktiv:= , 
	I_bFreigabeAuswerfen:= , 
	I_bSchrauberLogOn:= , 
	I_nMotorHersteller:= , 
	I_bHuettenSchr:= , 
	Q_bBusy=> 						stSKSSchrauberInOut_Vis_Schr_1.Q_bBusy, 
	Q_bDone=>						stSKSSchrauberInOut_Vis_Schr_1.Q_bDone ,	 
	Q_bError=>						stSKSSchrauberInOut_Vis_Schr_1.Q_bError , 
	Q_sPosZustand=> , 
	Q_bGrundstellungAktiv=> , 
	Q_bGrundstellungOk=> , 
	Q_bSchraubHub=> , 
	Q_bSchrAuswurf=> , 
	Q_bSchrHalt=> , 
	Q_bAxisReset=> , 
	Q_nErrorId=> 					stSKSSchrauberInOut_Vis_Schr_1.Q_nErrorId, 
	Q_bDrehmomentFehler=> 			stSKSSchrauberInOut_Vis_Schr_1.Q_bDrehmomentFehler, 
	Q_nStep=> 						stSKSSchrauberInOut_Vis_Schr_1.Q_nStep,
	Q_strStep=> , 
	Q_sStatus=> 					stSKSSchrauberInOut_Vis_Schr_1.Q_sStatus, 
	IQ_fbObjSchlauch:= 				objSchlauch, 
	IQ_stMeldung:= 					stAchsMeldung);
	
(*=============================================================================================*)	
(* Schlauch belegung *)
objSchlauch.I_bSchlauchBelegt		:=	stSKSSchrauberInOut_Vis_Schr_1.I_bSchlauchBelegt;
objSchlauch.I_bSchrauberBelegt		:=	stSKSSchrauberInOut_Vis_Schr_1.I_bSchrauberBelegt;
objSchlauch.I_bTasteVereinzelung	:=	stSKSSchrauberInOut_Vis_Schr_1.I_bVereinzelungStart;
objSchlauch.I_bSchrAuswurfStart		:=	stSKSSchrauberInOut_Vis_Schr_1.I_bAuswurfStart;

(*=============================================================================================*)	
(* Visu Übergabe *)
stSKSSchrauberInOut_Vis_Schr_1.Q_nActVelo	:=	arrNcAchsen[cAxis1261_Schrauber1].fVeloIstwert;
stSKSSchrauberInOut_Vis_Schr_1.Q_nActPos	:=	arrNcAchsen[cAxis1261_Schrauber1].fPosIstwert;
stSKSSchrauberInOut_Vis_Schr_1.Q_nActDepth	:=	arrNcAchsen[cEnc03_Schrauber1].fPosIstwert;


(*=============================================================================================*)	
(* Output Übergabe *)

bGVLVentil_1_Ausfahr:=		fbSchrauber_PnP_Original.Q_bSchraubHub;
bGVLVentil_1_Einfahr:=		NOT fbSchrauber_PnP_Original.Q_bSchraubHub;

bGVLVentil_2_Ausfahr:=		fbSchrauber_PnP_Original.Q_bSchrAuswurf;
bGVLVentil_2_Einfahr:=		NOT fbSchrauber_PnP_Original.Q_bSchrAuswurf;
END_ACTION

END_PROGRAM

// ---- POUs/SchrauberAblauf/FB_Schrauber_PnP.TcPOU
FUNCTION_BLOCK FB_Schrauber_PnP
// Version history:	
// 
// Bei Autoquit wird einmalig nach Zeit > T#0ms quittiert.
// Erst wieder nach erfolgreicher Bearbeitung kann ein Autoquit wieder aktiv werden.
// ( Vermeiden von Endlosschleifen von Fehlern )
// 
// Date          | Version    | created under        | Author          | Remark 
// ---------------------------------------------------------------------------------------- 
// ....          | ...        | ...                  | ...             | ...


VAR_INPUT
	
	I_bResetTeststation				: BOOL;		(* Hinzugefügt für Testaufbau im Steuerungstechniker Büro um den Baustein zu Quittieren !!*)
	
	I_bTaktFrg						: BOOL;
	I_bTaktStop						: BOOL;
	I_bAuto							: BOOL;
	I_bHand							: BOOL;
	I_bQuittFehler					: BOOL;
	I_bGrundstellung				: BOOL;
	I_bSchutzbereichOK			: BOOL;

	I_sSourceBeschreibung		: STRING;
	I_sPosBeschreibung			: STRING := 'Schrauber';

	I_bTaktStart					: BOOL;	(*Start Schienenschrauben*)
	I_bTaktStartHalb				: BOOL;	(*Start Schraube halb rein für z.B. Metalltravere*)

	I_bGrdstlgSchrEinh			: BOOL;
	I_bZustellZylAusgef			: BOOL;

	I_fSchraubTiefeAuswurf		: LREAL;

	I_fTiefentoleranzPositiv	: LREAL:=1;	(* Z.B. 3 bedeutet, dass von Solltiefe bis + 3mm wir im Ziel liegen *)
	I_fTiefentoleranzNegativ	: LREAL:=0.5;	(* Z.B. 3 bedeutet, dass von Solltiefe bis - 3mm wir im Ziel liegen *)
	I_nAchsId						: INT;
	I_nEncId							: INT;

	I_stParam						: ST_ParamSKSServoschrauber;

	I_tAutoQuit					: TIME :=T#0MS; (*default nicht aktiv -> 0ms *)
	
	I_bSchraubeNachschiessen	: BOOL;
	I_bReferenzfahrtAktiv		: BOOL;

	I_bFreigabeAuswerfen			: BOOL;
	
	I_sDateipfad					: STRING;
	I_bSchrauberLogOn				: BOOL;	// Umbennen in I_bSchrauberAbwahl

	I_nMotorHersteller			: INT; //0: BRC; 1: Beckhoff
	
	//Umbau Weber --> Boellhoff-/Huettenhoelscherschrauber
	I_bHuettenSchr					: BOOL := FALSE;

END_VAR

VAR_OUTPUT
	Q_bBusy						: BOOL;
	Q_bDone						: BOOL;
	Q_bError						: BOOL;

	Q_sPosZustand				: STRING := '';
	Q_bGrundstellungAktiv	: BOOL;
	Q_bGrundstellungOk		: BOOL;

	Q_bSchraubHub				: BOOL;
	Q_bSchrAuswurf				: BOOL;
	Q_bSchrHalt					: BOOL;
	Q_nTorque					: INT:=300;
	Q_bAxisReset				: BOOL;
	Q_nErrorId					: INT;
	Q_bDrehmomentFehler		: BOOL;
	Q_bTuerFreigabe			: BOOL;
	
	Q_nStep						: INT;
	Q_strStep					: STRING;
	
	Q_bModuloBetrArt			: BOOL;

	Q_sStatus					: STRING(255);	//Informationen zu dem aktuellen Ablaufschritt
END_VAR
VAR_IN_OUT
	IQ_fbObjSchlauch			: FB_Obj_IOSchlauch;				// Schlauch
	
	IQ_stMeldung				: ST_MeldServoSchrauber_1;		// Meldung

END_VAR
VAR
	objError_Schrauber		: FB_Obj_Error_Schrauber;

	bSchrAuswurfStart			: BOOL;
	bSchraubHub					: BOOL;
	bSchrAuswurf				: BOOL;
	
	bModuloBetrArt				: BOOL;
	
	fSchraubTiefeIst			: LREAL;
	arrDrehmomentIst			: ARRAY [0..10] OF LREAL;
	fDrehmomentIstMittel		: LREAL;
	tonAnlauf					: TON;
	tonStillstandAchse		: TON;
	tonStillstandVorschub	: TON;
	tonStillstVorschubDelay	: TON;
	fIstPosAchseAlt			: LREAL;
	fIstPosVorschubAlt		: LREAL;
	bStillstandAchse			: BOOL;
	bStillstandVorschub		: BOOL;
	nFehlerSchrittMerker		: INT;
	nFehlerZaehler				: INT;
	tonVerzStillstand			: TON;
	fReduzGeschwFaktor		: LREAL:= 0.025;	(* Reduzierter Geschwindigkeitsfaktur *)

	rtrigReset					: R_TRIG;
	bReset						: BOOL;
	bAchsreset					: BOOL;

	bAutoquitAktiv				: BOOL;
	tonAutoquit					: TON;
	tonTimeOver1				: TON;

	idx							: INT;

(* Schrittkette Grund*)
	nStepGrund  				: INT;
	nOldStepGrund				: INT;
	tonTimeOverGrund			: TON;

(* Schrittkette Auto*)
	nStep  						: INT;
	sStep							: STRING;
	nOldStep						: INT;
	tonDelay1					: TON;
	
	tonSchraubtakt				: TON;
	timeSchraubtakt			: TIME;
	arrLetzteTiefe				: ARRAY[0..100] OF LREAL;
	arrLetzteFehler			: ARRAY[0..100] OF LREAL;
	arrLetzteMomente			: ARRAY[0..100] OF LREAL;
	arrLetzteSchraubzeit		: ARRAY[0..100] OF TIME;
	ftrigStep60					: F_TRIG;
	bSchraubtest				: BOOL;
	nTestmoment					: UINT:=320;

	tonTimeOutSchrauber				: TON;
	nAnzahlSchraubspitzenKlemmer	: DINT;
	tonNotPosiFrg: TON;
	rtrigStep70: R_TRIG;
	ftrigStep70: F_TRIG;
	rtrigStepError: R_TRIG;
	
	fbMittelwert			: FB_Mittelwert;
	
	
	fSchraubTiefeIstTest				: LREAL;
	nTiefeBeimAufsetzen				: LREAL;
	bTiefeBeimAufsetzenOK			: BOOL;

	//Log
	fbStepHistory						: FB_StepHistory;

	fbLogToFile							: FB_LogFile_Schrauber;
	rtrigStueckzaehler				: R_TRIG;
	nStueckzaehler						: INT;
	rtrigSchrauberfehler				: R_TRIG;
	nTestStep1: INT;
	nTestStep2: INT;
	nTestStep3: INT;
END_VAR

	(* Reset *)
	rtrigReset(
		CLK:=IQ_fbObjSchlauch.I_bTasteNachruetteln);
		
	bReset:=rtrigReset.Q
			AND NOT (nStep = 10 OR nStep = 90)
			OR I_bResetTeststation;(* Hinzugefügt für Testaufbau im Steuerungstechniker Büro um den Baustein zu Quittieren !!*)

	a_Ablauf();
	e_Error();
	l_Log();
	o_Output();


	fReduzGeschwFaktor		:= 0.005;	(* Reduzierter Geschwindigkeitsfaktur *)

ACTION a_Ablauf:
IF NOT bReset THEN
	CASE nStep OF
	/////////////////////////////////////////////
	0: sStep												:='Setzen_Init';
	
		bSchraubHub										:= FALSE;
		bSchrAuswurf									:= FALSE;
		bAutoquitAktiv 								:= FALSE;
		bSchraubtest									:= FALSE;
		arrNcAchsen[I_nAchsId].stEinAusG.Q_nSignalsteuerwort.1	:= FALSE;
		tonNotPosiFrg(IN:=FALSE);

		IF I_bTaktFrg
		 AND NOT I_bGrundstellung THEN
			nStep := 10;
		END_IF

	/////////////////////////////////////////////
	10: sStep											:='Start';
	
		nFehlerSchrittMerker							:= 0;
		bTiefeBeimAufsetzenOK						:= FALSE;
		bModuloBetrArt									:= TRUE;

		tonNotPosiFrg(IN:=(NOT arrNcAchsen[I_nAchsId].stAuftrg.bPTP_PosiFrg
								AND arrNcAchsen[I_nAchsId].stEinAusG.I_nDCStatusword.13) // Am Regler steht ein Fehler an
								OR arrNcAchsen[I_nAchsId].bNcFehler,PT:=T#10S);

		bAchsreset :=
					tonNotPosiFrg.Q
					AND bTakt2langsam;

		IF NOT I_bReferenzfahrtAktiv
		THEN
			arrNcAchsen[I_nAchsId].stEinAusG.Q_nSignalsteuerwort.1			:= FALSE;
			arrNcAchsen[I_nAchsId].stGrdfkt.bIstw_setz	:= FALSE;
			arrStartAusf[I_nAchsId].I_bAchseZurArbP		:= FALSE;
		END_IF

		IF I_bSchraubeNachschiessen
		THEN
			IQ_fbObjSchlauch.I_bSchrauberBelegt:= FALSE;
		END_IF

		//AuswerfenStart
		IF (bSchrAuswurfStart
			OR IQ_fbObjSchlauch.I_bSchrAuswurfStart
			OR IQ_fbObjSchlauch.I_bTasteVereinzelung)
			AND NOT I_bTaktStop
		THEN
			IQ_fbObjSchlauch.I_bSchrAuswurfStart :=
			bSchrAuswurfStart := FALSE;
			tonTimeOver1(IN:=FALSE);
			nStep := 200;
			bAchsreset											:= FALSE;

		//Nachladen
		ELSIF NOT IQ_fbObjSchlauch.I_bSchrauberBelegt
			AND IQ_fbObjSchlauch.I_bSchlauchBelegt
			AND NOT I_bQuittFehler
			AND NOT I_bTaktStop
			THEN
				IF I_bHuettenSchr
				THEN
					tonTimeOver1(IN := TRUE, PT := t#0ms);
					bSchrAuswurf:=FALSE;
					
					//Warten bis Schrauberstange oben
					IF tonTimeOver1.Q
					THEN
						tonTimeOver1(IN := FALSE);
						nStep := 11;
					END_IF
				ELSE
					bSchrAuswurf:=TRUE;
					nStep := 11;
				END_IF
				bAchsreset											:= FALSE;

		//SetzenStart	-	Schienenschraube
		ELSIF IQ_fbObjSchlauch.I_bSchrauberBelegt
			AND I_bTaktStart
			AND NOT I_bTaktStop
			AND NOT I_bTaktStartHalb
			AND arrNcAchsen[I_nAchsId].stAuftrg.bPTP_PosiFrg
			AND I_bTaktFrg
			AND NOT I_bQuittFehler
			OR bSchraubtest
			THEN
				arrNcAchsen[I_nAchsId].stEinAusG.Q_nSignalsteuerwort.1					:= TRUE;
				arrNcAchsen[I_nAchsId].stGrdfkt.bIstw_setz			:= TRUE;
				arrNcAchsen[I_nAchsId].stGrdfkt.fIstSetzwert			:= 0;
				Q_nTorque														:= 3000;
				Q_bDrehmomentFehler 											:= FALSE;
         	
				bAchsreset:=FALSE;
				nStep 															:= 20;

		//SetzenStart	-	Einzelschraube halb rein für z.B. Metalltraver
		ELSIF IQ_fbObjSchlauch.I_bSchrauberBelegt
			AND NOT I_bTaktStart
			AND I_bTaktStartHalb
			AND NOT I_bTaktStop
			AND arrNcAchsen[I_nAchsId].stAuftrg.bPTP_PosiFrg
			AND I_bTaktFrg
			AND NOT I_bQuittFehler
			THEN
				arrNcAchsen[I_nAchsId].stEinAusG.Q_nSignalsteuerwort.1					:= TRUE;
				arrNcAchsen[I_nAchsId].stGrdfkt.bIstw_setz			:= TRUE;
				arrNcAchsen[I_nAchsId].stGrdfkt.fIstSetzwert			:= 0;
				Q_nTorque														:= 3000;

			IF bSchraubtest
			THEN
				Q_nTorque:= nTestmoment;
			END_IF

			bAchsreset:=FALSE;
			nStep 	:= 20;

		END_IF

	/////////////////////////////////////////
	11: sStep		:='Nachladen';

		IF (IQ_fbObjSchlauch.I_bSchrauberBelegt
			OR IQ_fbObjSchlauch.I_bTasteVereinzelung)
			AND NOT IQ_fbObjSchlauch.I_bNachladenaktiv

		THEN
			bSchrAuswurf	:= FALSE;
			tonTimeOver1(IN:= FALSE);
			nStep 			:= 12;
		END_IF
		
	/////////////////////////////////////////
	12: sStep		:='Nachladen - Warten bis Schrauberstange oben';
		tonTimeOver1(IN:= TRUE, PT:= T#200MS);
		
		IF tonTimeOver1.Q
		THEN
			bSchrAuswurf	:= FALSE;
			nStep 			:= 10;
		END_IF	

	/////////////////////////////////////////
	// Schrauben Schubkastenschiene			
	/////////////////////////////////////////
	20: sStep		:='SetzenStart';

		IF IQ_fbObjSchlauch.I_bSchrauberBelegt
			AND (I_bTaktStart OR I_bTaktStartHalb)
			AND I_bTaktFrg
			AND NOT I_bQuittFehler
			OR bSchraubtest
		THEN
			tonTimeOver1(IN:=FALSE);
			nStep := 30;
		END_IF

	/////////////////////////////////////////
	30: sStep		:='Schraubhub_vor';
	
		tonTimeOver1(IN:=TRUE,PT:=I_stParam.tParam_ZeitdZustellhubSchr);
		bSchraubHub		:= TRUE;

		IF I_bTaktFrg
			AND (tonTimeOver1.Q
				OR I_bZustellZylAusgef)
		THEN
			tonTimeOver1(IN:=FALSE);
			tonTimeOutSchrauber(IN:=FALSE);
			nStep := 40;
		END_IF

	/////////////////////////////////////////
	40:sStep		:='Auswerfhub_vor';
	
		tonTimeOver1(IN:=TRUE,PT:=I_stParam.tParam_ZeitdSchraubhubSchr);
		tonTimeOutSchrauber(IN:=TRUE,PT:=I_stParam.tParam_ZeitdSchraubhubSchr+T#2S);
		nTiefeBeimAufsetzen :=	fSchraubTiefeIst;
		bSchrAuswurf	:= TRUE;

		IF F_Inbetween(
					I_fActualValue := nTiefeBeimAufsetzen,
					I_fMinimalValue := 10 - 5,	//Tiefe beim Ausetzen auf die Seite, vor dem Schrauben
					I_fMaximalValue := 10 + 5)	
		THEN
			bTiefeBeimAufsetzenOK:= TRUE;
		END_IF

		IF tonTimeOver1.Q
		AND I_bTaktFrg
		AND NOT bSchraubtest
		AND F_Inbetween(
								I_fActualValue 	:= fSchraubTiefeIst,
								I_fMinimalValue 	:= I_stParam.fParam_Sollschraubtiefe - 100,
								I_fMaximalValue 	:= I_stParam.fParam_Sollschraubtiefe)
		THEN
			tonTimeOver1(IN:=FALSE);
			bSchraubHub												:= FALSE;
			bSchrAuswurf											:= FALSE;
			arrNcAchsen[I_nAchsId].stGrdfkt.bIstw_setz  	:= FALSE;
			IQ_fbObjSchlauch.I_bSchrauberBelegt 			:= FALSE;
			nFehlerZaehler											:= nFehlerZaehler + 1;
			nStep 													:= -40;			// Schraube fehlt 

		ELSIF tonTimeOver1.Q
		AND I_bTaktFrg
		AND arrNcAchsen[I_nAchsId].stGrdfkt.bIstw_gesetz
		AND arrNcAchsen[I_nAchsId].stAuftrg.bPTP_PosiFrg
		AND ((fSchraubTiefeIst
				<= 15)(*den Schrauber erst starten, wenn er durch das Mundstück hindurch ist*)(*Wieder rausgenommen, da es hin und wieder zu Störungen führte da das bit nicht durch das Mundstück hindurch kommt*)
				OR tonTimeOutSchrauber.Q)
		THEN
			IF tonTimeOutSchrauber.Q 
			THEN
				nAnzahlSchraubspitzenKlemmer := nAnzahlSchraubspitzenKlemmer + 1;
			END_IF
				tonTimeOutSchrauber(IN:=FALSE);
				tonTimeOver1(IN:=FALSE);
				arrNcAchsen[I_nAchsId].stGrdfkt.bIstw_setz	:= FALSE;
				nStep 											:= 45;
		END_IF

	/////////////////////////////////////////					 
   45:sStep		:='Schraubmotor langsam einschalten';
	
		tonTimeOver1(IN:=TRUE,PT:=T#5S);		(* Achtung OLD 5s - Nur geändert um mehr zu sehen	*)
	 	
	   arrNcAchsen[I_nAchsId].stAuftrg.fPTP_Geschw			:= I_stParam.fStartDrehzahl;
	   arrNcAchsen[I_nAchsId].stAuftrg.ePTP_BuffMode		:= MC_Aborting;
	   arrStartAusf[I_nAchsId].I_bAchseZurArbP				:= I_bTaktFrg;
    
	   IF (arrNcAchsen[I_nAchsId].stStatus.bFaehrtPos
	 	AND(	(arrNcAchsen[I_nAchsId].stAuftrg.fPTP_Geschw*0.8)		// wenn Achse 80% der Geschwindigkeit erreicht wurde
	 		  > (arrNcAchsen[I_nAchsId].fVeloIstwert						// in % umrechnen
					/arrNcAchsen[I_nAchsId].stParam.fEilgGeschw
					* 100)))			  
	   THEN 
	   	arrStartAusf[I_nAchsId].I_bAchseZurArbP		:= FALSE;
		  	tonTimeOver1(IN:=FALSE);
	 	  	nStep		:= 50; 	  
	   ELSIF tonTimeOver1.Q
	   THEN
			tonTimeOver1(IN:=FALSE);
			nStep 											:= 70;
			nFehlerSchrittMerker							:= -45;
	   END_IF

	/////////////////////////////////////////
	50:sStep		:='Schraubmotor laeuft schnell';
	
		tonTimeOver1(IN:=TRUE,PT:=T#3S);
	   arrStartAusf[I_nAchsId].I_bAchseZurArbP				:= I_bTaktFrg;

		IF I_bTaktStart
			AND fSchraubTiefeIst
				< I_stParam.fSchraubTiefeSollDrehzahl
		THEN
			arrNcAchsen[I_nAchsId].stAuftrg.fPTP_Geschw			:= I_stParam.fParam_Solldrehzahl;
			arrNcAchsen[I_nAchsId].stAuftrg.ePTP_BuffMode		:= MC_BlendingNext;
			arrStartAusf[I_nAchsId].I_bAchseZurArbP				:= I_bTaktFrg;
			
			nStep 															:= 60;
		ELSIF I_bTaktStartHalb
		THEN
			arrNcAchsen[I_nAchsId].stAuftrg.fPTP_Geschw			:= I_stParam.fParam_Solldrehzahl * 0.5;
			arrNcAchsen[I_nAchsId].stAuftrg.ePTP_BuffMode		:= MC_BlendingNext;
			arrStartAusf[I_nAchsId].I_bAchseZurArbP				:= I_bTaktFrg;
			
			nStep 															:= 60;
		ELSIF tonTimeOver1.Q
		THEN
			tonTimeOver1(IN:=FALSE);
			nStep 											:= 70;
			nFehlerSchrittMerker							:= -50;
		END_IF


	/////////////////////////////////////////
	60:sStep		:='Tiefenabfrage';
	
		tonTimeOver1(IN:=TRUE,PT:=I_stParam.tParam_ZeitdSchraubTakt);

		arrStartAusf[I_nAchsId].I_bAchseZurArbP				:= I_bTaktFrg;
		fbMittelwert(I_bReset:= TRUE);

		IF (F_Inbetween(
							I_fActualValue 	:= fSchraubTiefeIst,
							I_fMinimalValue 	:= -10,
							I_fMaximalValue 	:= I_stParam.fParam_Sollschraubtiefe )
			 AND I_bTaktStart)
		OR
			(F_Inbetween(
							I_fActualValue 	:= fSchraubTiefeIst,
							I_fMinimalValue 	:= 0,
							I_fMaximalValue 	:= I_stParam.fParam_SollschraubtiefeHerdumbau)(*Schraube nur "halb" rein*)
			 AND I_bTaktStartHalb)

			THEN
				//Drehzahlreduzierung um eine höhere Drehmomentgenauigkeit zu erreichen (letzter Stand 4% über soll)
				arrNcAchsen[I_nAchsId].stAuftrg.fPTP_Geschw		:= I_stParam.fParam_Solldrehzahl * 0.12;
				nStep 										 	:= 65;
				tonTimeOver1(IN:=FALSE);
		END_IF

		tonTimeOver1(IN:=TRUE,PT:=T#3000MS);
		IF tonTimeOver1.Q 
			AND tonDelay1.ET > T#3000MS
		THEN
			// Nicht O.K.: Tiefe nicht erreicht, 
			nStep 											:= 70;
			nFehlerSchrittMerker							:= -60;
			tonTimeOver1(IN:=FALSE);
		END_IF

	/////////////////////////////////////////
	65:sStep		:='Drehmomentabfrage';

		fbMittelwert(
				I_bReset			:= FALSE,
				I_fAktlWert		:= ABS(arrNcAchsen[I_nAchsId].stEinAusG.I_nDrehmomentIstwert),
				I_nAnzWerte		:= 10);

//		IF fbMittelwert.Q_fMittelwert
		IF fDrehmomentIstMittel
			>= I_stParam.fParam_Sollmoment * 100 * 1.1 
		AND I_bTaktStart
			THEN
				nStep 											:= 70;
		END_IF

//		IF fbMittelwert.Q_fMittelwert
		IF fDrehmomentIstMittel
			>= I_stParam.fParam_Sollmoment * 100 * 0.1 // 10% vom Sollmoment
		AND I_bTaktStartHalb
			THEN
				nTestStep3 := 			nTestStep3 + 1;
				nStep 											:= 70;
		END_IF

		//Nicht O.K.: Drehmoment nicht erreicht 
		IF tonDelay1.ET > I_stParam.tParam_ZeitdSchraubTakt  
		THEN
			IF fbMittelwert.Q_fMittelwert
				>= (I_stParam.fParam_Sollmoment * 100 / 5)
				THEN
				nTestStep1 := 			nTestStep1 + 1;
				nStep 											:= 70;
				nFehlerSchrittMerker							:= -65;
			ELSE
				nTestStep2 := 			nTestStep2 + 1;
				nStep 											:= 70;
				nFehlerSchrittMerker							:= -65;
			END_IF
		END_IF

		// Nicht O.K.: Keine Schraube vorhanden 
		IF fSchraubTiefeIst
			<=  I_stParam.fParam_Sollschraubtiefe - 10
			AND NOT bTiefeBeimAufsetzenOK
			THEN
				nStep 											:= 70;
				nFehlerSchrittMerker							:= -61;
		END_IF

	/////////////////////////////////////////
	//Halt auf die Achse geben, damit der Schrauber nicht wieder anlaufen kann und anschließend Sollwert = Istwert setzen
	70:sStep			:='Schraubmotor_Halt';
	
		tonTimeOver1(IN:=TRUE,PT:=T#1000MS);

		arrStartAusf[I_nAchsId].I_bAchseStopPos	:= TRUE;

		IF tonTimeOver1.Q
			OR arrStartAusf[I_nAchsId].Q_bAchseGestPos											
			OR arrStartAusf[I_nAchsId].Q_bAchseInPos
		THEN
			tonTimeOver1(IN:=FALSE);
			arrStartAusf[I_nAchsId].I_bAchseZurArbP		:= FALSE;

			IQ_fbObjSchlauch.I_bSchrauberBelegt 			:= FALSE;

			Q_nTorque	 	:= 0;

			nStep														:= 75;
		END_IF

	/////////////////////////////////////////
	75:sStep		:='Warten bis der Motor still steht';
	
		tonTimeOver1(IN:=TRUE,PT:=T#2000MS);

		IF tonTimeOver1.Q
			OR arrNcAchsen[I_nAchsId].stStatus.bInStillst 
		THEN
			tonTimeOver1(IN:=FALSE);
			nStep 													:= 80;
		END_IF

	/////////////////////////////////////////
	80:sStep		:='Spindelhub heben um ein Seitenhochziehen zu vermeiden';
	
		tonTimeOver1(IN:=TRUE,PT:=I_stParam.tParam_ZeitdAuswurfSchr);
		bSchrAuswurf												:= FALSE;
		
		IF F_Inbetween(
						I_fActualValue := fSchraubTiefeIst,
						I_fMinimalValue := 80 - 10,
						I_fMaximalValue := 80 + 10 )
		THEN
			tonTimeOver1(IN:=FALSE);
			nStep := 85;
		ELSIF tonTimeOver1.Q 
		THEN
			tonTimeOver1(IN:=FALSE);
			bSchraubHub	:= FALSE;
		  	nStep := 90;
			nFehlerSchrittMerker							:= -80;
		END_IF

	/////////////////////////////////////////
	85:sStep		:='Scharaubhub heben';
	
		bSchraubHub	:= FALSE;
		nStep 		:= 90;
						
	/////////////////////////////////////////
	90:sStep	:='Zylinder_Zur_Grundstellung';
      
		IF I_bGrdstlgSchrEinh
		 AND I_bTaktFrg
		THEN
			arrNcAchsen[I_nAchsId].stEinAusG.Q_nSignalsteuerwort.2	:= TRUE;		// Antriebsgeführtes Referenzieren 
			bAchsreset										:= TRUE;
			nStep := 95;
		END_IF

	/////////////////////////////////////////
	95:sStep	:='Antriebsgeführtes Referenzieren';
	
   	bAchsreset										:= FALSE;
   
		IF arrNcAchsen[I_nAchsId].stEinAusG.I_nSignalstatuswort.0
			OR I_nMotorHersteller = 1
		THEN
			arrNcAchsen[I_nAchsId].stEinAusG.Q_nSignalsteuerwort.2	:= FALSE;		// Antriebsgeführtes Referenzieren 

			IF nFehlerSchrittMerker <> 0
			THEN
				nFehlerZaehler			:= nFehlerZaehler + 1;
				nStep 					:= nFehlerSchrittMerker;
				nFehlerSchrittMerker	:= 0;
			ELSE
				nStep := 100;
			END_IF
		END_IF

	/////////////////////////////////////////
	100:sStep		:='Setzen Ende';
	
		bSchraubtest := FALSE;
		IF NOT I_bTaktStart
			AND NOT I_bTaktStartHalb
		THEN
			Q_nTorque	 										:= 300;
			bAutoquitAktiv 									:= FALSE;
			bSchraubtest										:= FALSE;
			arrNcAchsen[I_nAchsId].stEinAusG.Q_nSignalsteuerwort.1		:= FALSE;
			arrStartAusf[I_nAchsId].I_bAchseZurArbP	:= FALSE;			
			nStep		:= 10;
		END_IF

	/////////////////////////////////////////
	// Auswerfen										
	/////////////////////////////////////////
	200:sStep		:='AuswerfenStart';
	
		tonTimeOver1(IN:=TRUE,PT:=T#10S);
		IF I_bTaktFrg
		AND I_bFreigabeAuswerfen
			 OR tonTimeOver1.Q
			THEN
			tonTimeOver1(IN:=FALSE);
			nStep := 205;
		END_IF

	/////////////////////////////////////////
	205: sStep		:='Schraubhub_vor';
	
		tonTimeOver1(IN:=TRUE,PT:=I_stParam.tParam_ZeitdZustellhubSchr);
		bSchraubHub		:= TRUE;

		IF I_bTaktFrg
			AND (tonTimeOver1.Q
				OR I_bZustellZylAusgef)
		THEN
			tonTimeOver1(IN:=FALSE);
			nStep := 210;
		END_IF

	/////////////////////////////////////////
	210:sStep		:='Auswerfhub_zur';
	
		tonTimeOver1(IN:=TRUE,PT:=I_stParam.tParam_ZeitdAuswurfSchr);

		bSchrAuswurf	:= TRUE;

		IF F_Inbetween(
						I_fActualValue 	:= fSchraubTiefeIst,
						I_fMinimalValue 	:= I_fSchraubTiefeAuswurf - 100,
						I_fMaximalValue 	:= I_fSchraubTiefeAuswurf + 1 )
		THEN
			nStep := 230;
		ELSIF tonTimeOver1.Q THEN
			tonTimeOver1(IN:=FALSE,PT:=T#500MS);
			bSchrAuswurf	:= FALSE;
			nStep := 215;
		END_IF

	/////////////////////////////////////////
	215:
	
		tonTimeOver1(IN:=TRUE,PT:=T#100MS);
		IF tonTimeOver1.Q THEN
			tonTimeOver1(IN:=FALSE);
			nStep := 220;
		END_IF

	/////////////////////////////////////////
	220:sStep		:='Auswerfhub_zur';

		tonTimeOver1(IN:=TRUE,PT:=I_stParam.tParam_ZeitdAuswurfSchr);
		bSchrAuswurf	:= TRUE;

		IF F_Inbetween(
						I_fActualValue := fSchraubTiefeIst,
						I_fMinimalValue := I_fSchraubTiefeAuswurf - 100,
						I_fMaximalValue := I_fSchraubTiefeAuswurf + 1 )
		THEN
			nStep := 230;
			tonTimeOver1(IN:=FALSE,PT:=T#500MS);
		ELSIF tonTimeOver1.Q THEN
			bSchrAuswurf	:= FALSE;
			bSchraubHub		:= FALSE;
			nStep := -210;
			tonTimeOver1(IN:=FALSE,PT:=T#500MS);
		END_IF

	/////////////////////////////////////////
	230:sStep		:='AuswerfenAktiv';
	
		IF I_bTaktFrg THEN
			nStep := 240;
		END_IF

	/////////////////////////////////////////
	240:sStep		:='Auswerfhub_vor';
	
		tonTimeOver1(IN:=TRUE,PT:=T#1000MS);
		bSchrAuswurf	:= FALSE;
		bSchraubHub		:= FALSE;

		IF NOT F_Inbetween(
						I_fActualValue := fSchraubTiefeIst,
						I_fMinimalValue := I_fSchraubTiefeAuswurf - 100,
						I_fMaximalValue := I_fSchraubTiefeAuswurf + 1 )
			AND NOT I_bZustellZylAusgef
		THEN
			nStep := 250;
			tonTimeOver1(IN:=FALSE,PT:=T#1000MS);
		ELSIF tonTimeOver1.Q THEN
			bSchrAuswurf	:= FALSE;
			bSchraubHub		:= FALSE;
			nStep := -210;
			tonTimeOver1(IN:=FALSE,PT:=T#1000MS);
		END_IF

	/////////////////////////////////////////
	250:sStep		:='AuswerfenEnde';
	
		Q_nErrorId	:= 0;
		IF I_bTaktFrg AND NOT IQ_fbObjSchlauch.I_bTasteVereinzelung THEN
			IQ_fbObjSchlauch.I_bSchrauberBelegt := FALSE;
			bAutoquitAktiv := FALSE;
			nStep := 10;
		END_IF

	/////////////////////////////////////////
	// ERROR 
	/////////////////////////////////////////
	-40:sStep		:='Schraube fehlt';
	
		Q_nErrorId	:= -40;
		IF I_bQuittFehler
			AND I_bGrdstlgSchrEinh
			THEN
			bAutoquitAktiv := tonAutoquit.Q;
			bSchrAuswurfStart := TRUE;
			nStep := 100;
		END_IF

	/////////////////////////////////////////
	-45:sStep		:='Langsame Geschwindigkeit wird nicht erreicht';
	
		Q_nErrorId	:= -45;
		IF I_bQuittFehler
			AND I_bGrdstlgSchrEinh
			THEN
			bAutoquitAktiv := tonAutoquit.Q;
			bSchrAuswurfStart := TRUE;
			nStep := 100;
		END_IF

	/////////////////////////////////////////
	-50:sStep		:='Schraubtiefe für Solldrehzahl wird nicht erreciht';
	
		Q_nErrorId	:= -50;
		IF I_bQuittFehler
			AND I_bGrdstlgSchrEinh
			THEN
			bAutoquitAktiv := tonAutoquit.Q;
			bSchrAuswurfStart := TRUE;
			nStep := 100;
		END_IF

	/////////////////////////////////////////
	-60:sStep		:='Tiefe wird nicht erreicht';
	
		Q_nErrorId	:= -60;
		Q_bDrehmomentFehler := TRUE;

		IF I_bQuittFehler
			AND I_bGrdstlgSchrEinh
			THEN
			bAutoquitAktiv := tonAutoquit.Q;
			bSchrAuswurfStart := TRUE;
			nStep := 100;
		END_IF

	/////////////////////////////////////////
	-61: sStep		:='Tiefe ueberschritten';
	
		Q_nErrorId	:= -61;
		IF I_bQuittFehler
			AND I_bGrdstlgSchrEinh
			THEN
			bAutoquitAktiv := tonAutoquit.Q;
			bSchrAuswurfStart := TRUE;
			nStep := 100;
		END_IF

	/////////////////////////////////////////
	-65:sStep		:='Drehmoment wird nicht erreicht';
	
		Q_nErrorId	:= -65;
		IF I_bQuittFehler
			AND I_bGrdstlgSchrEinh
			THEN
			bAutoquitAktiv := tonAutoquit.Q;
			bSchrAuswurfStart := TRUE;
			nStep := 100;
		END_IF

	/////////////////////////////////////////
	-80:sStep		:='Fehler beim heben/senken der Schrauberstange';
	
		Q_nErrorId	:= -80;
		IF I_bQuittFehler
			AND I_bGrdstlgSchrEinh
			THEN
			bAutoquitAktiv := tonAutoquit.Q;
			bSchrAuswurfStart := TRUE;
			nStep := 100;
		END_IF
		
	/////////////////////////////////////////
	-210:sStep		:='Fehler Auswerfen';
	
		Q_nErrorId	:= -210;
		IF I_bQuittFehler
			THEN
			bAutoquitAktiv := tonAutoquit.Q;
			bSchrAuswurfStart := TRUE;
			nStep := 240;
		END_IF

	END_CASE
ELSE

	nStep := 0;

END_IF

	/////////////////////////////////////////
	IF I_bGrundstellung THEN
		nStep := 0;
	END_IF
	
	/////////////////////////////////////////
	// Autoquit 
	tonAutoquit(IN:=(Q_bError AND I_tAutoQuit > T#0MS),PT:=I_tAutoQuit);

	/////////////////////////////////////////
	//
	Q_sPosZustand := F_PosZustand(I_sString:=I_sPosBeschreibung, I_nStep:=nStep, I_sStep:=sStep);


	/////////////////////////////////////////
	// Ist-Schraubtiefe 
	fSchraubTiefeIst:= arrNcAchsen[I_nEncId].fPosIstwert;

	/////////////////////////////////////////
	// Mittelwert des Drehmoments bilden, damit nicht ein kurzer Ausschlag gleich zuer Abschaltung führen könnte 
	IF nStep >= 65
		AND nStep <= 70
	THEN
		arrDrehmomentIst[0]:= ABS(arrNcAchsen[I_nAchsId].stEinAusG.I_nDrehmomentIstwert);
		FOR idx:= 10 TO 1 BY -1 DO
			arrDrehmomentIst[idx]:= arrDrehmomentIst[idx-1];
		END_FOR
			fDrehmomentIstMittel:=	(	arrDrehmomentIst[1]
											+	arrDrehmomentIst[2]
											+	arrDrehmomentIst[3]
											+	arrDrehmomentIst[4]
											+	arrDrehmomentIst[5]
											+	arrDrehmomentIst[6]
											+	arrDrehmomentIst[7]
											+	arrDrehmomentIst[8]
											+	arrDrehmomentIst[9]
											+	arrDrehmomentIst[10]	)
											/	10;
	ELSE
		fDrehmomentIstMittel := 0;
	END_IF

	/////////////////////////////////////////
	//Schraubzeit für eigene Diagnose speichern
	tonSchraubtakt(
				IN:= nStep = 60 OR nStep = 160 OR nStep = 65,
				PT:= T#100s);
	IF nStep = 60
	OR nStep = 160
	OR nStep = 65
	THEN
		timeSchraubtakt:= tonSchraubtakt.ET;
	END_IF

	/////////////////////////////////////////
	//Informationen zur letzten Isttiefe, Schraubfehlernummer und anstehende Moment, 
	//werden zur eigenen, internen Diagnose in einem Array gespreichert 
	ftrigStep70(CLK:= nStep = 70);
	rtrigStep70(CLK:= nStep = 70
							//AND nFehlerSchrittMerker<>0
							);

	IF rtrigStep70.Q
	THEN
		FOR idx:=100 TO 1 BY -1 DO
			arrLetzteTiefe[idx]			:= arrLetzteTiefe[idx-1];
			arrLetzteFehler[idx]			:= arrLetzteFehler[idx-1];
			arrLetzteMomente[idx]		:= arrLetzteMomente[idx-1];
			arrLetzteSchraubzeit[idx]	:= arrLetzteSchraubzeit[idx-1];
		END_FOR
		arrLetzteTiefe[0]			:= fSchraubTiefeIst;
		arrLetzteFehler[0]		:=	nFehlerSchrittMerker;
		arrLetzteMomente[0]		:= fDrehmomentIstMittel;
		arrLetzteSchraubzeit[0]	:= timeSchraubtakt;
	END_IF

	/////////////////////////////////////////
	//Verzögerung des Achssignals "Stillstand" 
	tonVerzStillstand(
				IN:= arrNcAchsen[I_nAchsId].stStatus.bInStillst,
				PT:= T#10MS);
	
	//Timer
	tonDelay1(IN:=nStep= nOldStep,PT:=T#1D);
	nOldStep:= nStep;		
	
	//History	
	fbStepHistory(
		I_nStep := nStep );
END_ACTION

ACTION e_Error:
	(* Fehler überarbeitet *)

	(* Fehler Nachladen, Schraube fehlt *)
	objError_Schrauber.I_fbFehlerNachladen(
		I_bAktiv := (nStep = -40) 
						);
	(* Langsame Geschwindigkeit wird nicht erreicht *)
	objError_Schrauber.I_fbFehlerLangsameGeschwindigkeit(
		I_bAktiv := (nStep = -45) 
						);
	(* Schraubtiefe für Solldrehzahl wird nicht erreicht *)
	objError_Schrauber.I_fbFehlerTiefeSolldrehzahl(
		I_bAktiv := (nStep = -50) 
						);
	(* Tiefe nicht erreicht *)
	objError_Schrauber.I_fbFehler_Tiefe(
		I_bAktiv := (nStep = -60)
						);						
	(* Tiefe überschritten *)
	objError_Schrauber.I_fbFehler_TiefeUeberschritten(
		I_bAktiv := (nStep = -61)
						);
	(* Drehmoment nicht erreicht*)
	objError_Schrauber.I_fbFehler_Sollmoment(
		I_bAktiv := (nStep = -65)
						);
	(* Fehler beim heben/senken der Schrauberstange*)
	objError_Schrauber.I_fbFehler_Schrauberstange(
		I_bAktiv := (nStep = -80)
						);
	(* Fehler beim Auswerfen *)
	objError_Schrauber.I_fbFehlerAuswurf(
		I_bAktiv := (nStep = -210)
						);
	(* Fehler allgemein *)
	Q_bError	:= nStep<0
					AND NOT I_bSchrauberLogOn;
	
	
	IQ_stMeldung.bMeldFehlNachladen  					:= objError_Schrauber.I_fbFehlerNachladen.I_bAktiv
																		AND NOT I_bSchrauberLogOn;
	IQ_stMeldung.bMeldFehlLangsameGeschwindigkeit	:= objError_Schrauber.I_fbFehlerLangsameGeschwindigkeit.I_bAktiv
																		AND NOT I_bSchrauberLogOn;
	IQ_stMeldung.bMeldFehlTiefeSolldrehzahl			:= objError_Schrauber.I_fbFehlerTiefeSolldrehzahl.I_bAktiv
																		AND NOT I_bSchrauberLogOn;
	IQ_stMeldung.bMeldFehlSollTiefe						:= objError_Schrauber.I_fbFehler_Tiefe.I_bAktiv
																		AND NOT I_bSchrauberLogOn;
	IQ_stMeldung.bMeldFehlSollTiefeUebers				:= objError_Schrauber.I_fbFehler_TiefeUeberschritten.I_bAktiv
																		AND NOT I_bSchrauberLogOn;
	IQ_stMeldung.bMeldFehlSollDrehmom					:= objError_Schrauber.I_fbFehler_Sollmoment.I_bAktiv
																		AND NOT I_bSchrauberLogOn;
	IQ_stMeldung.bMeldFehlSchrauberstange				:= objError_Schrauber.I_fbFehler_Schrauberstange.I_bAktiv
																		AND NOT I_bSchrauberLogOn;
	IQ_stMeldung.bMeldFehlAuswerfen						:= objError_Schrauber.I_fbFehlerAuswurf.I_bAktiv
																		AND NOT I_bSchrauberLogOn;

	IQ_stMeldung.sName 		:= I_sPosBeschreibung;
	IQ_stMeldung.SourceName := I_sSourceBeschreibung;
END_ACTION

ACTION l_Log:
	//Stückzähler
	rtrigStueckzaehler(clk:= Q_bDone);
	IF rtrigStueckzaehler.Q
	THEN
		nStueckzaehler := nStueckzaehler + 1;
	END_IF
		
	//Log
	rtrigSchrauberfehler(clk:= nStep < 0
										AND I_stParam.bLogAnwahl);
   
	fbLogToFile(
		I_bStart				:= rtrigSchrauberfehler.Q,
		I_sDateipfad		:= I_sDateipfad,
		I_sDateiname		:= I_sPosBeschreibung,
		I_sUeberschrift	:= 'Timestamp;Anzahl;Schraubzeit;Drehmoment;Schraubtiefe;Barcode;Fehlermeldung;$R',
		
		I_bFehler1			:= objError_Schrauber.I_fbFehler_Schrauberstange.I_bAktiv,
		I_bFehler2			:= objError_Schrauber.I_fbFehler_Sollmoment.I_bAktiv,
		I_bFehler3			:= objError_Schrauber.I_fbFehler_Tiefe.I_bAktiv,
		I_bFehler4			:= objError_Schrauber.I_fbFehler_TiefeUeberschritten.I_bAktiv,
		I_bFehler5			:= objError_Schrauber.I_fbFehlerAuswurf.I_bAktiv,
		I_bFehler6			:= objError_Schrauber.I_fbFehlerLangsameGeschwindigkeit.I_bAktiv,
		I_bFehler7			:= objError_Schrauber.I_fbFehlerNachladen.I_bAktiv,
		I_bFehler8			:= objError_Schrauber.I_fbFehlerTiefeSolldrehzahl.I_bAktiv,
	               	   
		I_sFehler1			:= 'Fehler beim heben/senken der Schrauberstange',
		I_sFehler2			:= 'Fehler - Drehmoment wird nicht erreicht',
		I_sFehler3			:= 'Fehler - Tiefe wird nicht erreicht',
		I_sFehler4			:= 'Fehler - Tiefe ueberschritten',
		I_sFehler5			:= 'Fehler - Auswerfen',
		I_sFehler6			:= 'Fehler - Langsame Geschwindigkeit wird nicht erreicht',
		I_sFehler7			:= 'Fehler - Schraube fehlt',
		I_sFehler8			:= 'Fehler - Schraubtiefe für Solldrehzahl wird nicht erreicht',
   
		I_sBarcode			:= '',
   
		I_nAnzahlVerschraubungen := nStueckzaehler,
   
		I_tSchraubzeit		:= arrLetzteSchraubzeit[0],
		I_fDrehmoment		:= arrLetzteMomente[0],
		I_fSchraubtiefe	:= arrLetzteTiefe[0],
   	);		
   
	IF Q_bDone
	THEN
		fbLogToFile( I_bStart:= FALSE);
	END_IF
END_ACTION

ACTION o_Output:
	IQ_fbObjSchlauch.I_bSotiertopfEin :=
								I_bSchutzbereichOK AND NOT bReset
								AND (nStep = 11 OR nStep = 21);

	IQ_fbObjSchlauch.I_bFrgNachladen 	:=
								I_bSchutzbereichOK AND NOT bReset
								AND (nStep = 11);

	Q_bSchraubHub	:=		I_bSchutzbereichOK AND NOT bReset
								AND (bSchraubHub);

	Q_bSchrAuswurf	:=		I_bSchutzbereichOK AND NOT bReset
								AND (bSchrAuswurf);

	Q_bBusy			:= 	nStep <> 10 ;

	Q_bDone			:= 	nStep = 100 ;

	Q_bSchrHalt		:=		nStep = 70;			

	Q_bAxisReset	:=		bAchsreset ;

	Q_bTuerFreigabe:=
								nStep <= 10 ;
							
	Q_nStep 			:= 	nStep;
	Q_strStep		:= 	Q_strStep;
	
	Q_sStatus		:= Concat(INT_TO_STRING(nStep),CONCAT( ' - ', sStep));	

	(* ModuloBetrArt *)
	Q_bModuloBetrArt	:= bModuloBetrArt;
END_ACTION

END_FUNCTION_BLOCK

// ---- POUs/SchrauberAblauf/FB_Schrauber_PnP_Neu_1.TcPOU
// Überarbeitete Version mit vollständiger NC-Achsenintegration
(*
ABLAUFBESCHREIBUNG SERVOSCHRAUBER MIT NC-ACHSENANBINDUNG:

1. INITIALISIERUNG (Step 0)
   - Reset aller Ausgänge und Variablen
   - Prüfung der Grundbedingungen

2. STARTBEDINGUNGEN (Step 10)
   - Prüfung aller Freigaben und Sicherheitsbedingungen
   - Überprüfung des Schutzbereichs und NC-Status

3. ACHSEN-INITIALISIERUNG (Step 20)
   - Modulo-Betrieb aktivieren
   - Istwert auf 0 setzen
   - Drehmomentgrenzwert setzen

4. SCHRAUBHUB (Step 30)
   - Vorfahren des Schraubhubs
   - Überwachung des Zustellzylinders

5. DREHZAHLRAMPE (Step 45)
   - Kontrollierte Beschleunigung
   - Überwachung der erreichten Geschwindigkeit

6. HAUPTSCHRAUBVORGANG (Step 50/60)
   - Überwachung von Drehmoment und Tiefe
   - Geschwindigkeitsanpassung je nach Tiefe

7. DREHMOMENTÜBERWACHUNG (Step 65)
   - Mittelwertbildung des Drehmoments
   - Behandlung der vier Schraubfälle

8. ACHSEN-STOPP (Step 70)
   - Kontrolliertes Stoppen der Achse
   - Warten auf Stillstand

9. ABSCHLUSS (Step 80-95)
   - Rückfahrt in Grundstellung
   - Referenzierung bei Bedarf

10. FEHLERBEHANDLUNG (Step -1)
    - Zentrale Fehlerbehandlung
    - Achsen-Reset bei Bedarf
*)
FUNCTION_BLOCK FB_Schrauber_PnP_Neu_1
VAR_INPUT
	I_bResetTeststation				: BOOL;		(* Hinzugefügt für Testaufbau im Steuerungstechniker Büro um den Baustein zu Quittieren !!*)
    // Grundlegende Steuerungseingänge
    I_bTaktFrg               : BOOL;          // Freigabe für Takt
    I_bTaktStop              : BOOL;          // Stopp des Takts
    I_bAuto                  : BOOL;          // Automatikbetrieb
    I_bHand                  : BOOL;          // Handbetrieb
    I_bQuittFehler          : BOOL;          // Fehlerquittierung
    I_bGrundstellung        : BOOL;          // Grundstellungsanforderung
    I_bSchutzbereichOK      : BOOL;          // Schutzbereich freigegeben

    // Prozesseingänge
    I_bTaktStart            : BOOL;          // Start Schraubvorgang
    I_bTaktStartHalb        : BOOL;          // Start Halbschraubvorgang
    I_bGrdstlgSchrEinh      : BOOL;          // Grundstellung Schraubeinheit
    I_bZustellZylAusgef     : BOOL;          // Zustellzylinder ausgefahren

    // Parameter
    I_fSchraubTiefeAuswurf  : LREAL;         // Auswurftiefe
    I_fTiefentoleranzPos    : LREAL := 1.0;  // Positive Tiefentoleranz
    I_fTiefentoleranzNeg    : LREAL := 0.5;  // Negative Tiefentoleranz
    I_nAchsId               : INT;           // Achsen-ID für Schraubmotor
    I_nEncId                : INT;           // Encoder-ID für Tiefenmessung
    I_stParam               : ST_ParamSKSServoschrauber; // Parameter
    I_tAutoQuit             : TIME := T#0MS; // Automatische Quittierzeit
    
    // Steuerungseingänge
    I_bSchraubeNachschiessen: BOOL;          // Nachschiessen aktiv
    I_bReferenzfahrtAktiv   : BOOL;          // Referenzfahrt aktiv
    I_bFreigabeAuswerfen    : BOOL;          // Freigabe Auswerfen
    I_bSchrauberLogOn       : BOOL;          // Schrauber Logging aktiv
    I_nMotorHersteller      : INT;           // Motorhersteller (0:BRC, 1:Beckhoff)
    I_bHuettenSchr          : BOOL := FALSE; // Hüttenhölscher Schrauber aktiv
END_VAR

VAR_OUTPUT
    // Statusausgänge
    Q_bBusy                 : BOOL;          // Baustein aktiv
    Q_bDone                 : BOOL;          // Vorgang abgeschlossen
    Q_bError                : BOOL;          // Fehler aufgetreten
    Q_sPosZustand          : STRING := '';   // Aktueller Positionszustand
    Q_bGrundstellungAktiv  : BOOL;          // Grundstellung wird angefahren
    Q_bGrundstellungOk     : BOOL;          // Grundstellung erreicht
    
    // Prozessausgänge
    Q_bSchraubHub          : BOOL;           // Schraubhub aktiv
    Q_bSchrAuswurf         : BOOL;           // Auswurf aktiv
    Q_bSchrHalt            : BOOL;           // Schrauber gestoppt
    Q_bAxisReset           : BOOL;           // Achsreset angefordert
    Q_nErrorId             : INT;            // Fehler-ID
    Q_bDrehmomentFehler    : BOOL;           // Drehmomentfehler aufgetreten
    Q_nTorque			 	: INT:=300;
	
    // Debug und Status
    Q_nStep                : INT;            // Aktueller Schritt
    Q_strStep              : STRING;         // Schrittbeschreibung
    Q_sStatus              : STRING(255);    // Statustext
END_VAR

VAR_IN_OUT
    IQ_fbObjSchlauch       : FB_Obj_IOSchlauch;        // Schlauch
    IQ_stMeldung           : ST_MeldServoSchrauber_1;  // Meldung
END_VAR

VAR
    // Achsen-Istwerte (aus NC gelesen)
    fSchraubTiefeIst       : LREAL;          // Aktuelle Schraubtiefe
    fDrehmomentIst         : INT;            // Aktuelles Drehmoment in 0.1%
    fDrehzahlIst           : LREAL;          // Aktuelle Drehzahl
    
    // Sollwerte für Achse
    fSchraubTiefeSoll      : LREAL;          // Soll-Schraubtiefe
    fDrehzahlSoll          : LREAL;          // Solldrehzahl in %
    fDrehmomentGrenzwert   : LREAL;            // Drehmomentgrenzwert in 0.1%
    
    // Toleranzen und Grenzwerte
    fTiefenToleranz        : LREAL := 0.1;   // Toleranz für Tiefenmessung (mm)
    fMaxSpeed              : LREAL := 100.0; // Maximale Drehzahl (%)
    fReducedSpeed          : LREAL := 5.0;   // Reduzierte Drehzahl (%)
    fMaxTorque             : LREAL := 2000;    // Max Drehmoment (200.0%)
    fTorqueIncrement       : LREAL := 200;     // Drehmomenterhöhung (20.0%)
    
    // Rampenparameter
    tRampeHoch            : TIME := T#500MS; // Beschleunigungszeit
    fTiefeDrehzahlRed     : LREAL := 2.0;    // Abstand für Drehzahlreduzierung
    
    // Überwachungsvariablen
    fTiefenAenderung      : LREAL;           // Tiefenänderung über Zeit
    fLetzteTiefe          : LREAL;           // Letzte gemessene Tiefe
    nFehlerCounter        : INT;             // Fehlerzähler
    arrDrehmomentIst      : ARRAY [0..10] OF LREAL; // Array für Mittelwertbildung
    fDrehmomentIstMittel  : LREAL;             // Gemitteltes Drehmoment
    
    // Timer
    tonRampe              : TON;             // Timer für Rampensteuerung
    tonUeberwachung       : TON;             // Überwachungstimer
    tonStillstand         : TON;             // Stillstandsüberwachung
    tonGeschwindigkeit    : TON;             // Timer für Geschwindigkeitsüberwachung
    
    // Statusinformationen
    nSchraubFall          : INT;             // Aktueller Schraubfall (1-4)
    bSchraubphaseAktiv    : BOOL;            // Schraubphase aktiv
    bDrehmomentErreicht   : BOOL;            // Solldrehmoment erreicht
    bTiefenAenderungOK    : BOOL;            // Tiefenänderung im Toleranzbereich
    bAchseInitialisiert   : BOOL;            // Achse wurde initialisiert
    
    // Flankenmerker
    rtrigStart            : R_TRIG;          // Flanke für Start
    ftrigQuitt            : F_TRIG;          // Flanke für Quittierung
    
    // Index für Mittelwertbildung
    idx                   : INT;
END_VAR

// Flankenauswertung
rtrigStart(CLK:=I_bTaktStart);
ftrigQuitt(CLK:=I_bQuittFehler);

// Achsen-Istwerte kontinuierlich lesen
ReadAxisValues();

// Achsenfehler überwachen
CheckAxisErrors();

IF I_bResetTeststation
THEN
	Q_nStep := 0;
END_IF

// Hauptablauf
CASE Q_nStep OF
    
    // Initialisierung
    0: 
        Q_strStep := 'Initialisierung';
        ResetOutputs();
        IF I_bTaktFrg AND NOT I_bGrundstellung AND (I_bTaktStart OR rtrigStart.Q) THEN
            Q_nStep := 10;
            Q_bBusy := TRUE;
        END_IF

    // Start und Prüfung der Grundbedingungen
    10: 
        Q_strStep := 'Grundbedingungen prüfen';
		CheckStartConditions();
        IF CheckStartConditions() THEN
            // Parameter übernehmen
            fSchraubTiefeSoll := I_stParam.fParam_Sollschraubtiefe;
            fDrehmomentGrenzwert := I_stParam.fParam_Sollmoment; // 140.0% Startdrehmoment
            Q_nStep := 20;
        END_IF

    // Achsen-Initialisierung
    20:
        Q_strStep := 'Achse initialisieren';
        InitializeAxis();
        IF bAchseInitialisiert THEN
            Q_nStep := 30;
        END_IF

    // Schraubhub vorfahren
    30: 
        Q_strStep := 'Schraubhub vorfahren';
        Q_bSchraubHub := TRUE;
        tonUeberwachung(IN:=TRUE, PT:=I_stParam.tParam_ZeitdSchraubhubSchr);
        IF I_bZustellZylAusgef THEN
            tonUeberwachung(IN:=FALSE);
            Q_nStep := 40;
        ELSIF tonUeberwachung.Q THEN
            Q_bError := TRUE;
            Q_nErrorId := 80; // Fehler Schrauberstange
            Q_nStep := -1;
        END_IF

    // Auswerfhub vor (Tiefe prüfen)
    40:
        Q_strStep := 'Tiefe beim Aufsetzen prüfen';
        ExecuteTiefenPruefung();
        // Prüfen ob Schraube vorhanden
        IF fSchraubTiefeIst < (fSchraubTiefeSoll - 10.0) THEN
            nFehlerCounter := nFehlerCounter + 1;
            IF nFehlerCounter >= 2 THEN
                Q_bError := TRUE;
                Q_nErrorId := 40; // Schraube fehlt
                Q_nStep := -1;
            ELSE
                Q_nStep := 80; // Nochmal versuchen
            END_IF
        ELSE
            Q_nStep := 45;
        END_IF

    // Drehzahlrampe hochfahren
    45:
        Q_strStep := 'Drehzahl hochrampen';
        StartSpeedRamp();
        // Prüfen ob Geschwindigkeit erreicht
        IF CheckSpeedReached() THEN
            Q_nStep := 50;
        ELSIF tonGeschwindigkeit.Q THEN
            Q_bError := TRUE;
            Q_nErrorId := 45; // Geschwindigkeit nicht erreicht
            Q_nStep := -1;
        END_IF

    // Hauptschraubvorgang - schnelle Fahrt
    50:
        Q_strStep := 'Hauptschraubvorgang';
        ExecuteMainScrewing();
        // Prüfen ob Umschalttiefe erreicht
        IF fSchraubTiefeIst >= (I_stParam.fParam_Umschalttiefe - fTiefeDrehzahlRed) THEN
            Q_nStep := 60;
        END_IF

    // Tiefenabfrage und Drehzahlreduktion
    60:
        Q_strStep := 'Drehzahl reduzieren für Endposition';
        ReduceSpeed();
        IF CheckFinalPosition() THEN
            Q_nStep := 65;
        END_IF

    // Drehmomentüberwachung
    65:
        Q_strStep := 'Drehmomentüberwachung';
        MonitorTorque();
        DetermineSchraubfall();
        
        CASE nSchraubFall OF
            1: HandleCase1();
            2: HandleCase2();
            3: HandleCase3();
            4: HandleCase4();
        END_CASE
        
        // Prüfen ob Vorgang erfolgreich abgeschlossen
        IF CheckFinishConditions() THEN
            Q_nStep := 70;
        END_IF

    // Schraubvorgang beenden - Achse stoppen
    70:
        Q_strStep := 'Achse stoppen';
        StopAxis();
        IF arrNcAchsen[I_nAchsId].stStatus.bInStillst THEN
            Q_nStep := 75;
        END_IF

    // Warten und Stillstand sicherstellen
    75:
        Q_strStep := 'Warten auf Stillstand';
        tonStillstand(IN:=TRUE, PT:=T#100MS);
        IF tonStillstand.Q THEN
            tonStillstand(IN:=FALSE);
            Q_nStep := 80;
        END_IF

    // Schraubhub zurückfahren
    80:
        Q_strStep := 'Schraubhub zurück';
        Q_bSchraubHub := FALSE;
        Q_bSchrAuswurf := FALSE;
        tonUeberwachung(IN:=TRUE, PT:=T#500MS);
        IF tonUeberwachung.Q OR I_bGrdstlgSchrEinh THEN
            tonUeberwachung(IN:=FALSE);
            Q_nStep := 90;
        END_IF

    // Grundstellung anfahren
    90:
        Q_strStep := 'Grundstellung anfahren';
        ReturnToHome();
        IF I_bGrdstlgSchrEinh THEN
            Q_nStep := 95;
        END_IF

    // Referenzierung wenn nötig
    95:
        Q_strStep := 'Referenzierung';
        ReferenceAxis();
        IF arrNcAchsen[I_nAchsId].stEinAusG.I_nSignalstatuswort.0 OR I_nMotorHersteller = 1 THEN
            Q_bDone := TRUE;
            Q_bBusy := FALSE;
            Q_nStep := 0;
        END_IF

    // Fehlerbehandlung
    -1:
        Q_strStep := Q_sPosZustand;
        HandleError();
        IF ftrigQuitt.Q OR (I_tAutoQuit > T#0MS AND tonStillstand.Q) THEN
            ResetAxis();
            ResetOutputs();
            Q_nStep := 0;
        END_IF
END_CASE

// Timer für automatische Quittierung
IF Q_nStep = -1 AND I_tAutoQuit > T#0MS THEN
    tonStillstand(IN:=TRUE, PT:=I_tAutoQuit);
ELSE
    tonStillstand(IN:=FALSE);
END_IF

Q_nTorque	:=	LREAL_TO_INT(fDrehmomentGrenzwert);
// Grundstellung
Q_bGrundstellungOk := I_bGrdstlgSchrEinh AND Q_nStep = 0;

// Statusausgabe
Q_sStatus := CONCAT('Step ', INT_TO_STRING(Q_nStep));
Q_sStatus := CONCAT(Q_sStatus, ': ');
Q_sStatus := CONCAT(Q_sStatus, Q_strStep);

METHOD CheckAxisErrors
VAR
END_VAR
// NC-Fehler überwachen
IF arrNcAchsen[I_nAchsId].bNcFehler THEN
    Q_bError := TRUE;
    Q_nErrorId := 100; // NC-Fehler
    Q_strStep := CONCAT('NC-Fehler: ', DWORD_TO_STRING(arrNcAchsen[I_nAchsId].nFehlerNr));
END_IF

// DC-Status überwachen (Bit 13 = Antriebsfehler)
IF arrNcAchsen[I_nAchsId].stEinAusG.I_nDCStatusword.13 THEN
    Q_bError := TRUE;
    Q_nErrorId := 101; // Antriebsfehler
    Q_strStep := 'Antriebsfehler am Regler';
END_IF

// Positionsfreigabe verloren während Fahrt
IF Q_nStep >= 45 AND Q_nStep <= 70 THEN
    IF NOT arrNcAchsen[I_nAchsId].stAuftrg.bPTP_PosiFrg THEN
        Q_bError := TRUE;
        Q_nErrorId := 102; // Positionsfreigabe verloren
        Q_strStep := 'Positionsfreigabe verloren';
    END_IF
END_IF
END_METHOD

METHOD CheckFinalPosition : BOOL
VAR
END_VAR
// Prüfen ob Endposition erreicht wurde
CheckFinalPosition := fSchraubTiefeIst >= (fSchraubTiefeSoll - I_fTiefentoleranzNeg);

IF CheckFinalPosition THEN
    // Drehzahl auf Anzugsgeschwindigkeit reduzieren
    arrNcAchsen[I_nAchsId].stAuftrg.fPTP_Geschw := fReducedSpeed;
END_IF
END_METHOD

METHOD CheckFinishConditions : BOOL
VAR
    bDepthOK : BOOL;
    bTorqueOK : BOOL;
END_VAR
// Prüfen der Abschlussbedingungen
bDepthOK := (fSchraubTiefeIst >= (fSchraubTiefeSoll - I_fTiefentoleranzNeg)) AND 
            (fSchraubTiefeIst <= (fSchraubTiefeSoll + I_fTiefentoleranzPos));

bTorqueOK := (fDrehmomentIstMittel >= (fDrehmomentGrenzwert * 0.9)) AND 
             (fDrehmomentIstMittel <= fMaxTorque);

CheckFinishConditions := bDepthOK AND bTorqueOK;

IF CheckFinishConditions THEN
    Q_strStep := 'Schraubvorgang erfolgreich abgeschlossen';
END_IF
END_METHOD

METHOD CheckSpeedReached : BOOL
VAR
    fTargetSpeed : LREAL;
END_VAR
// Timer für Überwachung
tonGeschwindigkeit(IN:=TRUE, PT:=T#3S);

// Zielgeschwindigkeit berechnen (80% der Sollgeschwindigkeit)
fTargetSpeed := I_stParam.fStartDrehzahl * 0.8;

// Prüfen ob Geschwindigkeit erreicht wurde
CheckSpeedReached := arrNcAchsen[I_nAchsId].stStatus.bFaehrtPos AND
                     (arrNcAchsen[I_nAchsId].fVeloIstwert >= 
                      (fTargetSpeed * arrNcAchsen[I_nAchsId].stParam.fEilgGeschw / 100));

IF CheckSpeedReached THEN
    tonGeschwindigkeit(IN:=FALSE);
END_IF
END_METHOD

METHOD CheckStartConditions : BOOL
VAR
END_VAR
CheckStartConditions := 
    I_bTaktFrg AND
    NOT I_bTaktStop AND
    I_bSchutzbereichOK AND
    NOT Q_bError AND
    I_bGrdstlgSchrEinh AND  // Grundstellung muss erreicht sein
    arrNcAchsen[I_nAchsId].stAuftrg.bPTP_PosiFrg AND  // Achse hat Positionsfreigabe
    NOT arrNcAchsen[I_nAchsId].bNcFehler;  // Keine NC-Fehler
        
IF NOT CheckStartConditions THEN
    IF NOT I_bSchutzbereichOK THEN
        Q_strStep := 'Warte auf Schutzbereich';
    ELSIF NOT I_bGrdstlgSchrEinh THEN
        Q_strStep := 'Warte auf Grundstellung';
    ELSIF NOT arrNcAchsen[I_nAchsId].stAuftrg.bPTP_PosiFrg THEN
        Q_strStep := 'Warte auf Achsenfreigabe';
    ELSIF arrNcAchsen[I_nAchsId].bNcFehler THEN
        Q_strStep := 'NC-Fehler aktiv';
    END_IF
END_IF
END_METHOD

METHOD DetermineSchraubfall
VAR
END_VAR
// Bestimmung des aktuellen Schraubfalls
IF fSchraubTiefeIst < (fSchraubTiefeSoll - 10.0) THEN
    // Fall 4: Keine Schraube (große Tiefenabweichung)
    nSchraubFall := 4;
ELSIF bDrehmomentErreicht AND NOT bTiefenAenderungOK THEN
    // Fall 1: Drehmoment erreicht, aber Tiefe ändert sich noch
    IF fSchraubTiefeIst < fSchraubTiefeSoll THEN
        nSchraubFall := 1;
    ELSE
        nSchraubFall := 3; // Positive Toleranz
    END_IF
ELSIF bTiefenAenderungOK AND NOT bDrehmomentErreicht THEN
    // Fall 2: Tiefe erreicht, aber Drehmoment nicht
    nSchraubFall := 2;
ELSE
    // Normalfall
    nSchraubFall := 0;
END_IF
END_METHOD

METHOD ExecuteMainScrewing
VAR
END_VAR
// Hauptschraubvorgang mit voller Geschwindigkeit
arrNcAchsen[I_nAchsId].stAuftrg.fPTP_Geschw := I_stParam.fParam_Solldrehzahl;
arrNcAchsen[I_nAchsId].stAuftrg.ePTP_BuffMode := MC_BlendingNext;
arrStartAusf[I_nAchsId].I_bAchseZurArbP := I_bTaktFrg;

// Drehmomentüberwachung
bDrehmomentErreicht := fDrehmomentIstMittel >= fDrehmomentGrenzwert;

// Tiefenänderung überwachen
fTiefenAenderung := ABS(fSchraubTiefeIst - fLetzteTiefe);
bTiefenAenderungOK := fTiefenAenderung < 0.1; // Stillstand wenn < 0.1mm Änderung

// Speichern für nächsten Zyklus
fLetzteTiefe := fSchraubTiefeIst;

// Überwachung auf maximales Drehmoment
IF fDrehmomentIstMittel >= fMaxTorque THEN
    Q_bError := TRUE;
    Q_nErrorId := 65; // Drehmoment überschritten
    Q_nStep := -1;
END_IF
END_METHOD

METHOD ExecuteTiefenPruefung
VAR
END_VAR
// Auswerfhub aktivieren um Tiefe zu prüfen
Q_bSchrAuswurf := TRUE;
tonUeberwachung(IN:=TRUE, PT:=I_stParam.tParam_ZeitdSchraubhubSchr);

// Tiefe beim Aufsetzen speichern
IF tonUeberwachung.ET > T#100MS AND tonUeberwachung.ET < T#200MS THEN
    fLetzteTiefe := fSchraubTiefeIst;
END_IF

// Timeout-Überwachung
IF tonUeberwachung.Q THEN
    tonUeberwachung(IN:=FALSE);
    Q_bError := TRUE;
    Q_nErrorId := 80; // Fehler Schrauberstange
    Q_nStep := -1;
END_IF
END_METHOD

METHOD HandleCase1
VAR
END_VAR
// Fall 1: Negative Materialtoleranzen & Drehmoment erreicht
IF bDrehmomentErreicht AND NOT bTiefenAenderungOK THEN
    IF fDrehmomentGrenzwert < fMaxTorque THEN
        // Drehmoment schrittweise erhöhen
        fDrehmomentGrenzwert := fDrehmomentGrenzwert + fTorqueIncrement;
        arrNcAchsen[I_nAchsId].stEinAusG.Q_nDrehmomentGrenzwert := LREAL_TO_INT(fDrehmomentGrenzwert);
        arrNcAchsen[I_nAchsId].stAuftrg.fPTP_Geschw := fReducedSpeed;
        Q_strStep := 'Erhöhe Drehmoment';
    ELSE
        // Maximales Drehmoment erreicht
        Q_bError := TRUE;
        Q_nErrorId := 65;
        Q_nStep := -1;
    END_IF
END_IF
END_METHOD

METHOD HandleCase2
VAR
END_VAR
// Fall 2: Negative Materialtoleranzen & Solltiefe erreicht
IF bTiefenAenderungOK AND NOT bDrehmomentErreicht THEN
    IF fDrehmomentIstMittel < (fDrehmomentGrenzwert / 2) THEN
        // Drehmoment viel zu niedrig - Fehler
        Q_bError := TRUE;
        Q_nErrorId := 2;
        Q_strStep := 'Drehmoment nicht erreicht';
        Q_nStep := -1;
    ELSE
        // Leicht reduziertes Drehmoment akzeptabel
        arrNcAchsen[I_nAchsId].stAuftrg.fPTP_Geschw := fReducedSpeed;
    END_IF
END_IF
END_METHOD

METHOD HandleCase3
VAR
END_VAR
// Fall 3: Positive Materialtoleranzen
IF bDrehmomentErreicht AND NOT bTiefenAenderungOK THEN
    IF fDrehmomentGrenzwert < fMaxTorque THEN
        fDrehmomentGrenzwert := fDrehmomentGrenzwert + fTorqueIncrement;
        arrNcAchsen[I_nAchsId].stEinAusG.Q_nDrehmomentGrenzwert := LREAL_TO_INT(fDrehmomentGrenzwert);
        arrNcAchsen[I_nAchsId].stAuftrg.fPTP_Geschw := fReducedSpeed;
        Q_strStep := 'Positive Toleranz - Erhöhe Drehmoment';
    ELSE
        // Prüfen ob Tiefe trotzdem OK
        IF fSchraubTiefeIst >= (fSchraubTiefeSoll - I_fTiefentoleranzNeg) THEN
            // Akzeptabel
            Q_nStep := 70;
        ELSE
            Q_bError := TRUE;
            Q_nErrorId := 60; // Solltiefe nicht erreicht
            Q_nStep := -1;
        END_IF
    END_IF
END_IF
END_METHOD

METHOD HandleCase4
VAR
END_VAR
// Fall 4: Keine Schraube
IF fSchraubTiefeIst < (fSchraubTiefeSoll - 10.0) THEN
    nFehlerCounter := nFehlerCounter + 1;
    Q_strStep := CONCAT('Keine Schraube erkannt - Versuch ', INT_TO_STRING(nFehlerCounter));
    
    IF nFehlerCounter >= 2 THEN
        Q_bError := TRUE;
        Q_nErrorId := 40; // Schraube fehlt
        Q_strStep := 'Bitte Schraubsystem prüfen - Schraube fehlt';
        Q_nStep := -1;
    ELSE
        // Nochmal versuchen
        Q_nStep := 80; // Zurück zur Grundstellung
    END_IF
END_IF
END_METHOD

METHOD HandleError
VAR
END_VAR
// Fehlerbehandlung
Q_bError := TRUE;
Q_bSchraubHub := FALSE;
Q_bSchrAuswurf := FALSE;
Q_bSchrHalt := TRUE;

// Achse stoppen
arrStartAusf[I_nAchsId].I_bAchseStopPos := TRUE;
arrStartAusf[I_nAchsId].I_bAchseZurArbP := FALSE;

// Fehlerbeschreibung setzen
CASE Q_nErrorId OF
    2: // Drehmoment nicht erreicht
        Q_sPosZustand := 'Fehler: Drehmoment nicht erreicht';
        Q_bDrehmomentFehler := TRUE;
        
    40: // Schraube fehlt
        Q_sPosZustand := 'Fehler: Schraube fehlt';
        
    45: // Geschwindigkeit nicht erreicht
        Q_sPosZustand := 'Fehler: Geschwindigkeit nicht erreicht';
        
    60: // Solltiefe nicht erreicht
        Q_sPosZustand := 'Fehler: Solltiefe nicht erreicht';
        
    61: // Solltiefe überschritten
        Q_sPosZustand := 'Fehler: Solltiefe überschritten';
        
    65: // Drehmoment überschritten
        Q_sPosZustand := 'Fehler: Drehmoment überschritten';
        Q_bDrehmomentFehler := TRUE;
        
    80: // Fehler Schrauberstange
        Q_sPosZustand := 'Fehler: Schrauberstange/Zustellzylinder';
        
    100: // NC-Fehler
        Q_sPosZustand := 'Fehler: NC-Achse';
        
    101: // Antriebsfehler
        Q_sPosZustand := 'Fehler: Antrieb/Regler';
        
    102: // Positionsfreigabe verloren
        Q_sPosZustand := 'Fehler: Positionsfreigabe verloren';
        
    ELSE
        Q_sPosZustand := CONCAT('Fehler: Code ', INT_TO_STRING(Q_nErrorId));
END_CASE

// Meldungen setzen
UpdateErrorMessages();
END_METHOD

METHOD InitializeAxis
VAR
END_VAR
// Achse für Schraubvorgang initialisieren
bAchseInitialisiert := FALSE;

// Modulo-Betrieb aktivieren
arrNcAchsen[I_nAchsId].stEinAusG.Q_nSignalsteuerwort.1 := TRUE;

// Istwert auf 0 setzen
arrNcAchsen[I_nAchsId].stGrdfkt.bIstw_setz := TRUE;
arrNcAchsen[I_nAchsId].stGrdfkt.fIstSetzwert := 0;

// Drehmomentgrenzwert setzen
arrNcAchsen[I_nAchsId].stEinAusG.Q_nDrehmomentGrenzwert := LREAL_TO_INT(fDrehmomentGrenzwert);

// Warten bis Istwert gesetzt wurde
IF arrNcAchsen[I_nAchsId].stGrdfkt.bIstw_gesetz THEN
    arrNcAchsen[I_nAchsId].stGrdfkt.bIstw_setz := FALSE;
    bAchseInitialisiert := TRUE;
    Q_strStep := 'Achse initialisiert';
END_IF
END_METHOD

METHOD MonitorTorque
VAR
END_VAR
// Drehmoment-Mittelwertbildung für stabilere Messung
arrDrehmomentIst[0] := ABS(fDrehmomentIst);
FOR idx := 10 TO 1 BY -1 DO
    arrDrehmomentIst[idx] := arrDrehmomentIst[idx-1];
END_FOR

// Mittelwert berechnen
fDrehmomentIstMittel := 0;
FOR idx := 0 TO 10 DO
    fDrehmomentIstMittel := fDrehmomentIstMittel + arrDrehmomentIst[idx];
END_FOR
fDrehmomentIstMittel := fDrehmomentIstMittel / 11;

// Tiefenänderung überwachen
fTiefenAenderung := ABS(fSchraubTiefeIst - fLetzteTiefe);

// Überwachung des Drehmoments
IF fDrehmomentIstMittel >= fMaxTorque THEN
    Q_bError := TRUE;
    Q_nErrorId := 65; // Drehmoment zu hoch
    Q_nStep := -1;
ELSIF fSchraubTiefeIst >= fSchraubTiefeSoll AND 
      fDrehmomentIstMittel < (fDrehmomentGrenzwert / 2) THEN
    // Solltiefe erreicht aber Drehmoment viel zu niedrig
    Q_bError := TRUE;
    Q_nErrorId := 2; // Drehmoment zu niedrig
    Q_nStep := -1;
END_IF

// Überwachung auf Überschreitung der Solltiefe
IF fSchraubTiefeIst < (fSchraubTiefeSoll - I_fTiefentoleranzPos - 2.0) THEN
    Q_bError := TRUE;
    Q_nErrorId := 61; // Solltiefe überschritten
    Q_nStep := -1;
END_IF

fLetzteTiefe := fSchraubTiefeIst;
END_METHOD

METHOD ReadAxisValues
VAR
END_VAR
// Achsen-Istwerte aus NC lesen
fSchraubTiefeIst := arrNcAchsen[I_nEncId].fPosIstwert;
fDrehmomentIst := arrNcAchsen[I_nAchsId].stEinAusG.I_nDrehmomentIstwert;
fDrehzahlIst := arrNcAchsen[I_nAchsId].fVeloIstwert;
END_METHOD

METHOD ReduceSpeed
VAR
END_VAR
// Geschwindigkeit auf Anzugsgeschwindigkeit reduzieren
IF fSchraubTiefeIst >= (fSchraubTiefeSoll - fTiefeDrehzahlRed) THEN
    arrNcAchsen[I_nAchsId].stAuftrg.fPTP_Geschw := fReducedSpeed;
    Q_strStep := 'Reduziere Drehzahl für Endposition';
ELSE
    arrNcAchsen[I_nAchsId].stAuftrg.fPTP_Geschw := I_stParam.fParam_Solldrehzahl;
END_IF

// BufferMode für sanften Übergang
arrNcAchsen[I_nAchsId].stAuftrg.ePTP_BuffMode := MC_BlendingNext;
END_METHOD

METHOD ReferenceAxis
VAR
END_VAR
// Antriebsgeführtes Referenzieren
arrNcAchsen[I_nAchsId].stEinAusG.Q_nSignalsteuerwort.2 := TRUE;

// Warten auf Rückmeldung
IF arrNcAchsen[I_nAchsId].stEinAusG.I_nSignalstatuswort.0 THEN
    arrNcAchsen[I_nAchsId].stEinAusG.Q_nSignalsteuerwort.2 := FALSE;
    Q_strStep := 'Referenzierung abgeschlossen';
END_IF
END_METHOD

METHOD ResetAxis
VAR
END_VAR
// NC-Achse zurücksetzen
arrNcAchsen[I_nAchsId].stEinAusG.Q_nSignalsteuerwort.0 := TRUE; // Regler-Reset
arrNcAchsen[I_nAchsId].stGrdfkt.bReset_ausf := TRUE;

// Achse stoppen
arrStartAusf[I_nAchsId].I_bAchseStopPos := FALSE;
arrStartAusf[I_nAchsId].I_bAchseZurArbP := FALSE;

// Nach kurzer Zeit Reset zurücknehmen
tonStillstand(IN:=TRUE, PT:=T#100MS);
IF tonStillstand.Q THEN
    arrNcAchsen[I_nAchsId].stEinAusG.Q_nSignalsteuerwort.0 := FALSE;
    arrNcAchsen[I_nAchsId].stGrdfkt.bReset_ausf := FALSE;
    tonStillstand(IN:=FALSE);
END_IF

Q_bAxisReset := arrNcAchsen[I_nAchsId].stGrdfkt.bReset_ausf;
END_METHOD

METHOD ResetOutputs
VAR
END_VAR
// Reset aller Ausgänge
Q_bBusy := FALSE;
Q_bDone := FALSE;
Q_bError := FALSE;
Q_bSchraubHub := FALSE;
Q_bSchrAuswurf := FALSE;
Q_bSchrHalt := FALSE;
Q_bDrehmomentFehler := FALSE;
Q_bAxisReset := FALSE;
Q_nErrorId := 0;
Q_sPosZustand := '';
Q_strStep := 'Bereit';

// Reset interner Variablen
bDrehmomentErreicht := FALSE;
bTiefenAenderungOK := FALSE;
bAchseInitialisiert := FALSE;
nFehlerCounter := 0;
nSchraubFall := 0;
fLetzteTiefe := 0.0;
fTiefenAenderung := 0.0;
fDrehmomentIstMittel := 0;

// Timer zurücksetzen
tonRampe(IN:=FALSE);
tonUeberwachung(IN:=FALSE);
tonStillstand(IN:=FALSE);
tonGeschwindigkeit(IN:=FALSE);

// Arrays zurücksetzen
FOR idx := 0 TO 10 DO
    arrDrehmomentIst[idx] := 0;
END_FOR

// Achse zurücksetzen wenn nötig
IF arrNcAchsen[I_nAchsId].stEinAusG.Q_nSignalsteuerwort.1 THEN
    arrNcAchsen[I_nAchsId].stEinAusG.Q_nSignalsteuerwort.1 := FALSE;
END_IF
END_METHOD

METHOD ReturnToHome
VAR
END_VAR
// Zurück in Grundstellung
Q_bSchraubHub := FALSE;
Q_bSchrAuswurf := FALSE;
Q_bGrundstellungAktiv := TRUE;

// Achse in Grundstellung fahren (optional, abhängig von Mechanik)
IF NOT I_bGrdstlgSchrEinh THEN
    // Hier könnte eine Fahrt zur Grundstellung implementiert werden
    // z.B. arrNcAchsen[I_nAchsId].stAuftrg.fPTP_ZielPos := 0;
    Q_strStep := 'Fahre zur Grundstellung';
ELSE
    Q_bGrundstellungAktiv := FALSE;
    Q_strStep := 'Grundstellung erreicht';
END_IF
END_METHOD

METHOD StartSpeedRamp
VAR
END_VAR
// Drehzahlrampe starten
tonRampe(IN:=TRUE, PT:=tRampeHoch);

// Geschwindigkeit setzen
arrNcAchsen[I_nAchsId].stAuftrg.fPTP_Geschw := I_stParam.fStartDrehzahl;
arrNcAchsen[I_nAchsId].stAuftrg.ePTP_BuffMode := MC_Aborting;

// Achse starten
arrStartAusf[I_nAchsId].I_bAchseZurArbP := I_bTaktFrg;

// Lineare Rampe von Startdrehzahl auf Maximaldrehzahl
IF tonRampe.ET < tRampeHoch THEN
    fDrehzahlSoll := I_stParam.fStartDrehzahl + 
                     (I_stParam.fParam_Solldrehzahl - I_stParam.fStartDrehzahl) * 
                     TIME_TO_REAL(tonRampe.ET) / TIME_TO_REAL(tRampeHoch);
    arrNcAchsen[I_nAchsId].stAuftrg.fPTP_Geschw := fDrehzahlSoll;
ELSE
    arrNcAchsen[I_nAchsId].stAuftrg.fPTP_Geschw := I_stParam.fParam_Solldrehzahl;
    tonRampe(IN:=FALSE);
END_IF
END_METHOD

METHOD StopAxis
VAR
END_VAR
// Achse kontrolliert stoppen
arrStartAusf[I_nAchsId].I_bAchseStopPos := TRUE;
arrStartAusf[I_nAchsId].I_bAchseZurArbP := FALSE;

// Drehmomentgrenzwert auf 0 setzen
arrNcAchsen[I_nAchsId].stEinAusG.Q_nDrehmomentGrenzwert := 0;

// Warten auf Rückmeldung
IF arrStartAusf[I_nAchsId].Q_bAchseGestPos OR 
   arrStartAusf[I_nAchsId].Q_bAchseInPos OR
   arrNcAchsen[I_nAchsId].stStatus.bInStillst THEN
    Q_strStep := 'Achse gestoppt';
END_IF
END_METHOD

METHOD UpdateErrorMessages
VAR
END_VAR
// Meldungsstruktur aktualisieren
IQ_stMeldung.bMeldFehlNachladen := (Q_nErrorId = 40);
IQ_stMeldung.bMeldFehlLangsameGeschwindigkeit := (Q_nErrorId = 45);
IQ_stMeldung.bMeldFehlTiefeSolldrehzahl := FALSE; // Nicht mehr verwendet
IQ_stMeldung.bMeldFehlSollTiefe := (Q_nErrorId = 60);
IQ_stMeldung.bMeldFehlSollTiefeUebers := (Q_nErrorId = 61);
IQ_stMeldung.bMeldFehlSollDrehmom := (Q_nErrorId = 2) OR (Q_nErrorId = 65);
IQ_stMeldung.bMeldFehlSchrauberstange := (Q_nErrorId = 80);
IQ_stMeldung.bMeldFehlAuswerfen := FALSE; // Auswerflogik nicht implementiert

IQ_stMeldung.sName := 'Servoschrauber';
IQ_stMeldung.SourceName := 'FB_Schrauber_PnP_Neu';
END_METHOD

END_FUNCTION_BLOCK

// ---- POUs/Simulationsprogramm/FB_Schrauber_Simulation.TcPOU
(*
SIMULATIONSBAUSTEIN FÜR SERVOSCHRAUBER
=======================================
Simuliert die Hardware-Komponenten für den Schraubertest:
- NC-Achse (Drehmotor)
- Encoder (Tiefenmessung)
- Zustellzylinder
- 4 verschiedene Schraubfälle

SCHRAUBFÄLLE:
1. Negative Toleranz & Drehmoment erreicht
2. Negative Toleranz & Solltiefe erreicht  
3. Positive Toleranz
4. Keine Schraube
*)
FUNCTION_BLOCK FB_Schrauber_Simulation
VAR_INPUT
    // Steuerung
    I_bSimulationEnable     : BOOL;          // Simulation aktivieren
    I_bReset                : BOOL;          // Reset der Simulation
    I_nSimulatedCase        : INT := 0;      // Zu simulierender Fall (0=Normal, 1-4=Fehlerfälle)
    
    // Parameter für Simulation
    I_fSollTiefe            : LREAL := -5.0; // Solltiefe in mm
    I_fMaxDrehzahl          : LREAL := 3000; // Max Drehzahl in U/min
    I_fMaxDrehmoment        : LREAL := 2.0;  // Max Drehmoment in Nm
    
    // Eingänge vom Schrauber-FB
    I_bSchraubHub           : BOOL;          // Schraubhub-Befehl
    I_bSchrAuswurf          : BOOL;          // Auswurf-Befehl
    I_nAchsId               : INT;           // Achsen-ID
    I_nEncId                : INT;           // Encoder-ID
END_VAR

VAR_OUTPUT
    // Simulierte Hardware-Ausgänge
    Q_bZustellZylAusgef     : BOOL;          // Zustellzylinder ausgefahren
    Q_bGrdstlgSchrEinh      : BOOL;          // Grundstellung erreicht
    Q_bSchutzbereichOK      : BOOL := TRUE;  // Schutzbereich OK
    
    // Debug-Ausgänge
    Q_fSimTiefe             : LREAL;         // Aktuelle simulierte Tiefe
    Q_fSimDrehmoment        : LREAL;         // Aktuelles simuliertes Drehmoment
    Q_fSimDrehzahl          : LREAL;         // Aktuelle simulierte Drehzahl
    Q_sDebugInfo            : STRING(255);   // Debug-Information
END_VAR

VAR
    // Interne Simulationsvariablen
    fAchsPosition           : LREAL;         // Simulierte Achsposition (Winkel)
    fTiefe                  : LREAL;         // Simulierte Tiefe
    fDrehmoment             : LREAL;         // Simuliertes Drehmoment
    fDrehzahl               : LREAL;         // Simulierte Drehzahl
    fZielDrehzahl           : LREAL;         // Ziel-Drehzahl
    
    // Timer für Simulation
    tonZylinder             : TON;           // Timer für Zylinderbewegung
    tonTiefenSimulation     : TON;           // Timer für Tiefenänderung
    tonDrehmomentAufbau     : TON;           // Timer für Drehmomentaufbau
    
    // Zustandsvariablen
    bSchraubeVorhanden      : BOOL := TRUE;  // Schraube vorhanden
    bMaterialHart           : BOOL;          // Hartes Material (höheres Drehmoment)
    bMaterialWeich          : BOOL;          // Weiches Material (niedrigeres Drehmoment)
    nSimulationStep         : INT;           // Interner Simulationsschritt
    
    // Einfache Rampen-Variablen (ohne externe Library)
    fDrehzahlRampe          : LREAL;         // Rampen-Zwischenwert Drehzahl
    fDrehmomentRampe        : LREAL;         // Rampen-Zwischenwert Drehmoment
    fRampeBeschleunigung    : LREAL := 50.0; // Beschleunigung U/min pro Zyklus
    fRampeBremsung          : LREAL := 100.0;// Bremsung U/min pro Zyklus
    fDrehmomentAnstieg      : LREAL := 0.02; // Drehmomentanstieg Nm pro Zyklus
END_VAR

// Simulation nur wenn aktiviert
IF NOT I_bSimulationEnable THEN
    RETURN;
END_IF

// Reset-Logik
IF I_bReset THEN
    ResetSimulation();
    RETURN;
END_IF

